// TwinCAT 3 PLC project Felber
// ProgramVersion: 3.1.4024.0
// libraries:
//   EfficientIO Communicator, * (EfficientIO)
//   EfficientIO Energy Basic, * (EfficientIO)
//   Lynus Persistent Data V1, * (Lynus AG)
//   Lynus Standards, * (EfficientIO)
//   Tc2_BABasic, * (Beckhoff Automation GmbH)
//   Tc2_EtherCAT, * (Beckhoff Automation GmbH)
//   Tc2_Standard, * (Beckhoff Automation GmbH)
//   Tc2_System, * (Beckhoff Automation GmbH)
//   Tc2_Utilities, * (Beckhoff Automation GmbH)
//   Tc3_IPCDiag, * (Beckhoff Automation GmbH)
//   Tc3_Module, * (Beckhoff Automation GmbH)
// project tree:
//   DUTs/ struct_ADS_Felber.TcDUT
//   ENUMs/ E_State.TcDUT
//   / FastTask.TcTTO (not stored), MiddleTask.TcTTO, SlowTask.TcTTO (not stored)
//   FBs/EL3443_DPM/DUTs/ E_EL3443_DPM_Phase.TcDUT (not stored), E_EL3443_DPM_Total.TcDUT (not stored), MDP5001_341_7CD731EE.TcDUT, MDP5001_341_I_7CD731EE.TcDUT (not stored), MDP5001_341_O_7CD731EE.TcDUT (not stored), ST_EL3443_DPM_MUX_REAL.TcDUT, ST_EL3443_DPM_MUX_ULINT.TcDUT, ST_EL3443_DPM_StatusLx.TcDUT, ST_EL3443_DPM_StatusTotal.TcDUT, ST_EL3443_DPM_VariantLx.TcDUT (not stored), ST_EL3443_DPM_VariantTotal.TcDUT (not stored), ST_EL3443_DPM_VariantValues.TcDUT
//   FBs/EL3443_DPM/ FB_EL3443_DPM.TcPOU
//   FBs/EL3446 FW02 or higher/DUTs/ E_EL3446_Phase.TcDUT, MDP5001_342_066CA8C6.TcDUT (not stored), MDP5001_342_I_066CA8C6.TcDUT (not stored), MDP5001_342_O_066CA8C6.TcDUT (not stored), ST_EL3446_MUX_REAL.TcDUT (not stored), ST_EL3446_MUX_ULINT.TcDUT, ST_EL3446_StatusIx.TcDUT, ST_EL3446_VariantIx.TcDUT, ST_EL3446_VariantValues.TcDUT
//   FBs/EL3446 FW02 or higher/ FB_EL3446.TcPOU (not stored)
//   FBs/ FB_CoE_EL3446.TcPOU, FB_CoE_EL3443.TcPOU, FB_EM_Beckhoff_EL3443.TcPOU, FB_EM_Beckhoff_EL3446.TcPOU, FB_TimeSwitch_V2.TcPOU (not stored), prg_ReadDeviceName.TcPOU (not stored)
//   POUs/ prgComEffIO.TcPOU, prgEM.TcPOU (not stored), prgEMS.TcPOU, prgHW_v1.TcPOU (not stored), prgPersistent.TcPOU, prgRWEffIO.TcPOU (not stored), prgSystemTime.TcPOU (not stored), prgVarEffIO.TcPOU (not stored)

CONFIGURATION Felber
    RESOURCE PLC ON TwinCAT3
        TASK MiddleTask(INTERVAL := T#10ms, PRIORITY := 22);
        PROGRAM prgPersistent WITH MiddleTask : prgPersistent;
        PROGRAM prgSystemTime WITH MiddleTask : prgSystemTime;
        PROGRAM prgEM WITH MiddleTask : prgEM;
        PROGRAM prgEMS WITH MiddleTask : prgEMS;
    END_RESOURCE
END_CONFIGURATION

// ---- DUTs/struct_ADS_Felber.TcDUT
TYPE struct_ADS_Felber :
STRUCT
	int_liveCount		: INT;	
	
	// prgEM
	lr_RealPower_Grid			: LREAL;				
	lr_ApparentPower_Grid		: LREAL;				
	lr_ReactivePower_Grid		: LREAL;				
	lr_Frequency_Grid			: LREAL;				                                   
	lr_Voltage_L1N				: LREAL;				
	lr_Voltage_L2N				: LREAL;				
	lr_Voltage_L3N				: LREAL;				
	lr_Voltage_L1L2				: LREAL;				
	lr_Voltage_L2L3				: LREAL;				
	lr_Voltage_L3L1				: LREAL;				
 	lr_Current_L1				: LREAL;				
	lr_Current_L2				: LREAL;				
	lr_Current_L3				: LREAL;				
	lrPower_EM1					: LREAL;					
	lrPower_EM2					: LREAL;					
	lrPower_EM3					: LREAL;					
	lrPower_EM4					: LREAL;					
	lrPower_EM5					: LREAL;					
	lrPower_EM6					: LREAL;					
	lrPower_House				: LREAL;					
	lr_EnergyCounter_Grid		: LREAL;					
	lr_EnergyCounter_EM1		: LREAL;					
	lr_EnergyCounter_EM2		: LREAL;					
	lr_EnergyCounter_EM3		: LREAL;					
	lr_EnergyCounter_EM4		: LREAL;					
	lr_EnergyCounter_EM5		: LREAL;					
	lr_EnergyCounter_EM6		: LREAL;					
	lr_EnergyCounter_House		: LREAL;		

	// prgEMS
	b_Manual_On_CH1				: BOOL;						
	b_Manual_Off_CH1			: BOOL;						
	b_Manual_On_CH2				: BOOL;						
	b_Manual_Off_CH2			: BOOL;						
	b_Manual_On_CH3				: BOOL;						
	b_Manual_Off_CH3			: BOOL;						
	b_Manual_On_CH4				: BOOL;						
	b_Manual_Off_CH4			: BOOL;						
	b_Manual_On_CH5				: BOOL;						
	b_Manual_Off_CH5			: BOOL;						
	b_Manual_On_Coffee_CH6		: BOOL;				
	b_Manual_Off_Coffee_CH6		: BOOL;				
	b_Manual_On_Vent_CH7		: BOOL;				
	b_Manual_Off_Vent_CH7		: BOOL;			
	b_LoadOn_CH1				: BOOL;		
	b_LoadOn_CH2				: BOOL;			
	b_LoadOn_CH3				: BOOL;			
	b_LoadOn_CH4				: BOOL;			
	b_LoadOn_CH5				: BOOL;			
	b_LoadOn_CH6				: BOOL;			
	b_LoadOn_CH7				: BOOL;		
	byte_MoFr_Open_Hour			: BYTE;					
	byte_MoFr_Open_Minute		: BYTE;					
	byte_MoFr_Close_Hour		: BYTE;					
	byte_MoFr_Close_Minute		: BYTE;					
	byte_Sa_Open_Hour			: BYTE;					
	byte_Sa_Open_Minute			: BYTE;					
	byte_Sa_Close_Hour			: BYTE;					
	byte_Sa_Close_Minute		: BYTE;					
	byte_So_Open_Hour			: BYTE;					
	byte_So_Open_Minute			: BYTE;					
	byte_So_Close_Hour			: BYTE;					
	byte_So_Close_Minute		: BYTE;					
// offset CH1 in hours			                    
	b_Enable_Control_CH1		: BOOL;				
	real_Offset_Start_CH1		: REAL;				
	real_Offset_Stop_CH1		: REAL;				
// offset CH2 in hours			                    
	b_Enable_Control_CH2		: BOOL;				
	real_Offset_Start_CH2		: REAL;				
	real_Offset_Stop_CH2		: REAL;				
// offset CH3 in hours			                    
	b_Enable_Control_CH3		: BOOL;				
	real_Offset_Start_CH3		: REAL;				
	real_Offset_Stop_CH3		: REAL;				
// offset CH4 in hours			                    
	b_Enable_Control_CH4		: BOOL;				
	real_Offset_Start_CH4		: REAL;				
	real_Offset_Stop_CH4		: REAL;				
// offset CH5 in hours			                    
	b_Enable_Control_CH5		: BOOL;				
	real_Offset_Start_CH5		: REAL;				
	real_Offset_Stop_CH5		: REAL;				
// offset CH6 in hours			                    
	b_Enable_Control_Coffee_CH6	: BOOL;				
	real_Offset_Start_Coffee_CH6: REAL;				
	real_Offset_Stop_Coffee_CH6	: REAL;				
// offset CH7 in hours			                    
	b_Enable_Control_Vent_CH7	: BOOL;				
	real_Offset_Start_CH7		: REAL;				
	real_Offset_Stop_CH7		: REAL;				


                                  
			(*: REAL;			                        
			: REAL;                                     
			: REAL;			
			: REAL;			
			: REAL;
			: REAL;			
			: REAL;
			: REAL;			
*)

END_STRUCT
END_TYPE

// ---- ENUMs/E_State.TcDUT
{attribute 'qualified_only'}
TYPE E_State :
(
	Init := 0,
	ReadOnce,
	Error,
	Idle,
	Wait

	
);
END_TYPE

// ---- FBs/EL3443_DPM/DUTs/MDP5001_341_7CD731EE.TcDUT
TYPE MDP5001_341_7CD731EE :
STRUCT
	MDP5001_341_Input	: MDP5001_341_I_7CD731EE;
	MDP5001_341_Output	: MDP5001_341_O_7CD731EE;
END_STRUCT
END_TYPE

// ---- FBs/EL3443_DPM/DUTs/ST_EL3443_DPM_MUX_REAL.TcDUT
TYPE ST_EL3443_DPM_MUX_REAL :
STRUCT
    nSelector : UINT := E_EL3443_DPM_Phase.Error_INDEX_Not_Valid;
    fValueRef : REFERENCE TO REAL;
END_STRUCT
END_TYPE

// ---- FBs/EL3443_DPM/DUTs/ST_EL3443_DPM_MUX_ULINT.TcDUT
TYPE ST_EL3443_DPM_MUX_ULINT :
STRUCT
    nSelector : UINT := E_EL3443_DPM_Phase.Error_INDEX_Not_Valid;
    nValueRef : POINTER TO ULINT;
END_STRUCT
END_TYPE

// ---- FBs/EL3443_DPM/DUTs/ST_EL3443_DPM_StatusLx.TcDUT
TYPE ST_EL3443_DPM_StatusLx :
STRUCT
    bStatus_Voltage_Sign_Bit : BOOL;             //Voltage Sign Bit - Indicates the sign of the current sine wave voltage: 1 = U > 0V, 0 = U < 0V
    bStatus_Overvoltage : BOOL;                  //Overvoltage - Maximum measurable voltage is exceeded.
    bStatus_Overcurrent : BOOL;                  //Overcurrent - Maximum measurable current is exceeded.
    bStatus_Inaccurate_Voltage : BOOL;           //Inaccurate Voltage - The measured voltage value is smaller than the value entered in CoE object "F800:15 Inaccurate Threshold Voltage".
    bStatus_Inaccurate_Current : BOOL;           //Inaccurate Current - The measured current value is smaller than the value entered in CoE object "F800:16 Inaccurate Threshold Current".
    bStatus_Voltage_Guard_Warning : BOOL;        //Voltage Guard Warning - A warning limit of the voltage monitor has been breached.
    bStatus_Voltage_Guard_Error : BOOL;          //Voltage Guard Error - An error limit of the voltage monitor has been breached.
    bStatus_Current_Guard_Warning : BOOL;        //Voltage Current Warning - A warning limit of the Current monitor has been breached.
    bStatus_Current_Guard_Error : BOOL;          //Voltage Current Error - An error limit of the Current monitor has been breached.
    bStatus_TxPDO_Toggle : BOOL;                 //TxPDO Toggle - The TxPDO toggle is toggled by the slave when the data of the associated TxPDO is updated.
END_STRUCT
END_TYPE

// ---- FBs/EL3443_DPM/DUTs/ST_EL3443_DPM_StatusTotal.TcDUT
TYPE ST_EL3443_DPM_StatusTotal :
STRUCT
    bStatus_System_State : BOOL;                         //System State - Overall system state (as a logical disjunction of voltage guard errors, phase sequence, overvoltage, overcurrent and frequency guard errors)
    bStatus_Grid_Direction : BOOL;                       //Grid Direction - Phase sequence L1 - L2 - L3 correctly detected (with clockwise 3-phase mains)
    bStatus_Frequency_Guard_Warning : BOOL;              //Frequency Guard Warning - A warning limit of the frequency monitor has been breached.
    bStatus_Frequency_Guard_Error : BOOL;                //Frequency Guard Error - An error limit of the frequency monitor has been breached.
    bStatus_Neutral_Current_Guard_Warning : BOOL;        //Neutral Current Guard Warning - A warning limit of the neutral conductor current monitor has been breached.
    bStatus_Neutral_Current_Guard_Error : BOOL;          //Neutral Current Guard Error - An error limit of the neutral conductor current monitor has been breached.
    bStatus_Active_Power_Guard_Warning : BOOL;           //Active Power Guard Warning - A warning limit of the active power monitor has been breached.
    bStatus_Active_Power_Guard_Error : BOOL;             //Active Power Guard Error - An error limit of the active power monitor has been breached.
    bStatus_Apparent_Power_Guard_Warning : BOOL;         //Apparent Power Guard Warning - A warning limit of the apparent power monitor has been breached.
    bStatus_Apparent_Power_Guard_Error : BOOL;           //Apparent Power Guard Error - An error limit of the apparent power monitor has been breached.
    bStatus_Power_Quality_Guard_Warning : BOOL;          //Power Quality Guard Warning - A warning limit of the PQF monitor has been breached.
    bStatus_Power_Quality_Guard_Error : BOOL;            //Power Quality Guard Error - An error limit of the PQF monitor has been breached.
    bStatus_TxPDO_State : BOOL;                          //TxPDO State - TRUE for general error
    bStatus_TxPDO_Toggle : BOOL;                         //TxPDO Toggle - The TxPDO toggle is toggled by the slave when the data of the associated TxPDO is updated.
    fStatus_Power_Quality_Factor : REAL;                 //Power Quality Factor - Analog value of the voltage quality between 1.0 and 0 (see basic function principles - Power Quality Factor)
END_STRUCT                                              
END_TYPE

// ---- FBs/EL3443_DPM/DUTs/ST_EL3443_DPM_VariantValues.TcDUT
{attribute 'no-analysis'}
TYPE ST_EL3443_DPM_VariantValues :
STRUCT
	astLx 			: ARRAY[1..3] OF ST_EL3443_DPM_VariantLx;
	stTotal 		: ST_EL3443_DPM_VariantTotal;
END_STRUCT
END_TYPE

// ---- FBs/EL3446 FW02 or higher/DUTs/E_EL3446_Phase.TcDUT
(*This enum is equivalent to the selectors from the documentation " Confirmation of variable output values 1 - 4"*)
{attribute 'qualified_only'}
TYPE E_EL3446_Phase :
(
    nPhaseI1_OFFSET := 256,     //Offset Channel 1(Current I1). The offset is added to the base selector     
    nPhaseI2_OFFSET := 512,     //Offset Channel 2(Current I2). The offset is added to the base selector
    nPhaseI3_OFFSET := 768,     //Offset Channel 3(Current I3). The offset is added to the base selector
    nPhaseI4_OFFSET := 1024,    //Offset Channel 4(Current I1). The offset is added to the base selector     
    nPhaseI5_OFFSET := 1280,    //Offset Channel 5(Current I2). The offset is added to the base selector
    nPhaseI6_OFFSET := 1536,    //Offset Channel 6(Current I3). The offset is added to the base selector
    
    
    U_RMS:= 1,                  // [V] (Real Selector: 1 (Examp.: 257 = 1 + 256 for ch. 1)) RMS value of the voltage
    I_RMS:= 8,                  // [A] (Real Selector: 8) RMS value of the current 
	Frequency:= 17,             // [Hz] (Real Selector: 17) Frequency of this phase
    Phi:= 21,                   // [°] (Real Selector: 21) Phase angle of the fundamental wave
    Cos_phi:= 22,               // [-] (Real Selector: 22) Cosine of the fundamental wave phase angle
    Power_Factor:= 23,          // [-] (Real Selector: 23) Power factor
    P:= 26,                     // [W] (Real Selector: 26) Active power
	(*available with FW02 and higher*) Pavg := 27,                 // [W] (Real Selector: 27) Average active power during the last interval
	(*available with FW02 and higher*) Pmin := 28,                 // [W] (Real Selector: 28) Minimum active power in the last interval
	(*available with FW02 and higher*) Pmax := 29,                 // [W] (Real Selector: 29) Maximum active power in the last interval
	Pfund:= 30,					// [W] (Real Selector: 30) Fundamental wave active power in the last interval
    S_:= 32,                    // [VA] (Real Selector: 32) Apparent power
	(*available with FW02 and higher*) Savg := 33,                 // [W] (Real Selector: 33) Average apparent power during the last interval
	(*available with FW02 and higher*) Smin := 34,                 // [W] (Real Selector: 34) Minimum apparent power in the last interval
	(*available with FW02 and higher*) Smax := 35,                 // [W] (Real Selector: 35) Maximum apparent power in the last interval
	Sfund:= 36,					// [VA] (Real Selector: 36) Fundamental wave apparent power in the last interval
    Q:= 38,                     // [Var] (Real Selector: 38) Reactive power
	(*available with FW02 and higher*) Qavg := 39,                 // [W] (Real Selector: 39) Average reactive power during the last interval
	(*available with FW02 and higher*) Qmin := 40,                 // [W] (Real Selector: 40) Minimum reactive power in the last interval
	(*available with FW02 and higher*) Qmax := 41,                 // [W] (Real Selector: 41) Maximum reactive power in the last interval
	Qfund:= 42,					// [Var] (Real Selector: 36) Fundamental wave reactive power in the last interval
    EP:= 45,                    // [mhW] (UINT Selector: 45) Recorded active energy
    EP_pos:= 46,                // [mhW] (UINT Selector: 46) Received active energy
    EP_neg:= 47,                // [mhW] (UINT Selector: 47) Supplied active energy
	EP_interval:= 48, 			// [mhW] (UINT Selector: 48) Recorded active energy in the last interval
	EP_pos_interval:= 49, 		// [mhW] (UINT Selector: 49) Received active energy in the last interval
	EP_neg_interval:= 50, 		// [mhW] (UINT Selector: 50) Supplied active energy in the last interval
    ES:= 51,                    // [mhW] (UINT Selector: 51) Apparent energy
    ES_pos:= 52,                // [mhW] (UINT Selector: 52) Apparent energy
    ES_neg:= 53,                // [mhW] (UINT Selector: 53) Apparent energy
	ES_interval:= 54, 			// [mhW] (UINT Selector: 54) Apparent energy in the last interval
	ES_pos_interval:= 55, 		// [mhW] (UINT Selector: 55) Apparent energy in the last interval
	ES_neg_interval:= 56, 		// [mhW] (UINT Selector: 56) Apparent energy in the last interval
    EQ_:= 57,                   // [mhW] (UINT Selector: 57) Reactive energy
    EQ_pos:= 58,                // [mhW] (UINT Selector: 58) Reactive energy
    EQ_neg:= 59,                // [mhW] (UINT Selector: 59) Reactive energy
	EQ_interval:= 60, 			// [mhW] (UINT Selector: 60) Reactive energy in the last interval
	EQ_pos_interval:= 61, 		// [mhW] (UINT Selector: 62) Reactive energy in the last interval
	EQ_neg_interval:= 62, 		// [mhW] (UINT Selector: 63) Reactive energy in the last interval
    THD_U:= 95,                 // [-] (Real Selector: 95) "Total Harmonic Distortion" is the distortion factor of the voltage. It indicates the ratio of the harmonic components of an oscillation relative to its fundamental.
    RMS_fund_U:= 98,            // [V] (Real Selector: 98) Amplitude of the fundamental wave
	THD_I:= 165,                // [-] (Real Selector: 165) "Total Harmonic Distortion" is the distortion factor of the current. It indicates the ratio of the harmonic components of an oscillation relative to its fundamental.
    RMS_fund_I:= 168,           // [A] (Real Selector: 168) Amplitude of the fundamental wave
    (*available with FW02 and higher*) F_Ref_I:= 169,              // [Hz] (Real Selector: 169) Reference frequency of the current harmonic: Specifies the underlying fundamental frequency, e.g.: 50 or 60 Hz.
    Harmonics_I := 170,         // [% of the fundamental wave] (Real Selector: 170-211) 0 => DC component, 1 => fundamental wave, 2=> 2nd harmonic, 3=> 3rd harmonic
    Error_INDEX_Not_Valid:= 255 // [-] (Real Selector: 255) Error message: The selected index is not available.
)UINT;
END_TYPE

// ---- FBs/EL3446 FW02 or higher/DUTs/ST_EL3446_MUX_ULINT.TcDUT
TYPE ST_EL3446_MUX_ULINT :
STRUCT
    nSelector : UINT := E_EL3446_Phase.Error_INDEX_Not_Valid;
    nValueRef : POINTER TO ULINT;
END_STRUCT
END_TYPE

// ---- FBs/EL3446 FW02 or higher/DUTs/ST_EL3446_StatusIx.TcDUT
TYPE ST_EL3446_StatusIx :
STRUCT
	bOvercurrent : BOOL;                    //Overcurrent - Maximum measurable current is exceeded.
	bInaccurate_Current : BOOL;             //Inaccurate Current - The measured current value is outside the limits for the current entered in CoE object 0x80n2
	bCurrent_Guard_Warning : BOOL;          //Current Guard Warning - The measured current value is outside the warning limits entered in the CoE objects 0x80n2:06 and 0x80n2:07
	bCurrent_Guard_Error : BOOL;            //Current Guard Error - The measured current value is outside the error limits entered in the CoE objects 0x80n2:05 and 0x80n2:08
	bApparent_Power_Guard_Warning : BOOL;   //Apparent Power Guard Warning - The value for the apparent power is outside the warning limits entered in the CoE objects 0x80n2:0A and 0x80n2:0B
	bApparent_Power_Guard_Error : BOOL;     //Apparent Power Guard Error - The value for the apparent power is outside the error limits for the current entered in the CoE objects 0x80n2:09 and 0x80n2:0C
	bActive_Power_Guard_Warning : BOOL;     //Active Power Guard Warning - The value for active power is outside the warning limits entered in the CoE objects 0x80n2:0E and 0x80n2:0F
	bActive_Power_Guard_Error : BOOL;       //Active Power Guard Error - The value for active power is outside the error limits for the current entered in CoE objects 0x80n2:0D and 0x80n2:10
	bReactive_Power_Guard_Warning : BOOL;   //Reactive Power Guard Warning - The value for the reactive power is outside the warning limits entered in the CoE objects 0x80n2:12 and 0x80n2:13
	bReactive_Power_Guard_Error : BOOL;     //Reactive Power Guard Error - The value for the reactive power is outside the error limits for the current entered in the CoE objects 0x80n2:11 and 0x80n2:14
	bDPM_Inaccurate : BOOL;                 //DPM Inaccurate
	bDPM_Timeout : BOOL;                    //DPM Toggl e- The DPM toggle is toggled by the slave when the DPM data has been updated.
	bTxPDO_Toggle : BOOL;                   //TxPDO Toggle - The TxPDO toggle is toggled by the slave when the data of the associated TxPDO has been updated.
	fCurrent : REAL;                        //Current - Actual measured current value
	fActive_Power : REAL;                   //Active Power - Actually measured active power
	fApparent_Power : REAL;                 //Apparent Power - Actual measured apparent power
	fReactive_Power_Fundamental : REAL;     //Reactive Power Fundamental - Balanced reactive power fundamental oscillation
	nActive_Energy : DINT;                  //Active Energy - Actually measured active energy
END_STRUCT
END_TYPE

// ---- FBs/EL3446 FW02 or higher/DUTs/ST_EL3446_VariantIx.TcDUT
TYPE ST_EL3446_VariantIx :
STRUCT
    fU_RMS : REAL;// [V] (Real Selector: 1 (Examp.: 257 = 1 + 256 for ch. 1)) RMS value of the voltage
    fI_RMS : REAL;// [A] (Real Selector: 8) RMS value of the current
    fFrequency : REAL;// [Hz] (Real Selector: 17) Frequency of this phase
    fPhi : REAL;// [°] (Real Selector: 21) Phase angle of the fundamental wave
    fCOS_phi : REAL;// [-] (Real Selector: 22) Cosine of the fundamental wave phase angle
    fPower_Factor : REAL;// [-] (Real Selector: 23) Power factor
    fP : REAL;// [W] (Real Selector: 26) Active power
	(*available with FW02 and higher*) fPavg : REAL;						// [W] (Real Selector: 27) Average active power during the last interval
    (*available with FW02 and higher*) fPmin : REAL;						// [W] (Real Selector: 28) Minimum active power in the last interval
    (*available with FW02 and higher*) fPmax : REAL;						// [W] (Real Selector: 29) Maximum active power in the last interval
	fPfund : REAL;// [W] (Real Selector: 30) Fundamental wave active power in the last interval
	fS : REAL;// [VA] (Real Selector: 32) Apparent power
	(*available with FW02 and higher*) fSavg : REAL;						// [VA] (Real Selector: 33) Average apparent power during the last interval
    (*available with FW02 and higher*) fSmin : REAL;						// [VA] (Real Selector: 34) Minimum apparent power in last interval
   	(*available with FW02 and higher*) fSmax : REAL;						// [VA] (Real Selector: 35) Minimum apparent power in last interval
    fSfund : REAL;// [VA] (Real Selector: 36) Fundamental wave apparent power in the last interval
    fQ : REAL;// [Var] (Real Selector: 38) Reactive power
	(*available with FW02 and higher*) fQavg : REAL;						// [Var] (Real Selector: 39) Average reactive power average during the last interval
    (*available with FW02 and higher*) fQmin : REAL;						// [Var] (Real Selector: 40) Minimum reactive power in the last interval
    (*available with FW02 and higher*) fQmax : REAL;						// [Var] (Real Selector: 41) Maximum reactive power in the last interval
    fQfund : REAL;// [Var] (Real Selector: 42) Fundamental wave reactive power in the last interval
    nEP : LINT;// [mhW] (LINT Selector: 45) Recorded active energy
    nEP_pos : ULINT;// [mhW] (UINT Selector: 46) Received active energy
    nEP_neg : ULINT;// [mhW] (UINT Selector: 47) Supplied active energy
	nEP_interval : LINT;// [mhW] (LINT Selector: 48) Recorded active energy in the last interval
	nEP_pos_interval : ULINT;// [mhW] (UINT Selector: 49) Received active energy in the last interval
	nEP_neg_interval : ULINT;// [mhW] (UINT Selector: 50) Supplied active energy in the last interval
    nES : LINT;// [mhW] (LINT Selector: 51) Apparent energy
    nES_pos : ULINT;// [mhW] (UINT Selector: 52) Apparent energy
    nES_neg : ULINT;// [mhW] (UINT Selector: 53) Apparent energy
	nES_interval : LINT;// [mhW] (LINT Selector: 54) Apparent energy in the last interval
	nES_pos_interval : ULINT;// [mhW] (UINT Selector: 55) Apparent energy in the last interval
	nES_neg_interval : ULINT;// [mhW] (UINT Selector: 56) Apparent energy in the last interval
    nEQ : LINT;// [mhW] (LINT Selector: 57) Reactive energy
    nEQ_pos : ULINT;// [mhW] (UINT Selector: 58) Reactive energy
    nEQ_neg : ULINT;// [mhW] (UINT Selector: 59) Reactive energy
	nEQ_interval : LINT;// [mhW] (LINT Selector: 60) Reactive energy in the last interval
	nEQ_pos_interval : ULINT;// [mhW] (UINT Selector: 62) Reactive energy in the last interval
	nEQ_neg_interval : ULINT;// [mhW] (UINT Selector: 63) Reactive energy in the last interval
    fTHD_U : REAL;// [-] (Real Selector: 95) "Total Harmonic Distortion" is the distortion factor of the voltage. It indicates the ratio of the harmonic components of an oscillation relative to its fundamental.
    fRMS_fund_U : REAL;// [V] (Real Selector: 98) Amplitude of the fundamental wave
    fTHD_I : REAL;// [-] (Real Selector: 165) "Total Harmonic Distortion" is the distortion factor of the current. It indicates the ratio of the harmonic components of an oscillation relative to its fundamental.
    fRMS_fund_I : REAL;// [A] (Real Selector: 168) Amplitude of the fundamental wave
    (*available with FW02 and higher*) fF_Ref_I : REAL;// [Hz] (Real Selector: 169) Reference frequency of the current harmonic: Specifies the underlying fundamental frequency, e.g.: 50 or 60 Hz.
    fHarmonics_I : ARRAY [0..41] OF REAL;// [% of the fundamental wave] (Real Selector: 170-211) 0 => DC component, 1 => fundamental wave, 2=> 2nd harmonic, 3=> 3rd harmonic
END_STRUCT
END_TYPE

// ---- FBs/EL3446 FW02 or higher/DUTs/ST_EL3446_VariantValues.TcDUT
{attribute 'no-analysis'}
TYPE ST_EL3446_VariantValues :
STRUCT
	astIx 			: ARRAY[1..6] OF ST_EL3446_VariantIx;
END_STRUCT
END_TYPE

// ---- POUs/prgPersistent.TcPOU
PROGRAM prgPersistent
VAR
	fbUSV		: FB_WritePersistentData_CX81xx;

	fb_Reboot		: NT_reboot;
	m_Reboot		: BOOL:=FALSE;
END_VAR

fbUSV(
	eSaveModeData:= eUSVSaveMode.eSaveWhenPowerfail, 
	bLoadPersistentDataOk=> , 
	bPowerFailDetect=> , 
	bError=> , 
	bySaveProcess=> , 
	dwStorageLast24h=> , 
	udiErrorCode=> );
	
	
		
fb_Reboot(	netid := '',
			delay := 2,
			start := m_Reboot);

END_PROGRAM

// ---- POUs/prgEMS.TcPOU
PROGRAM prgEMS
VAR
	FB_TimeSwitch_CH1: FB_TimeSwitch_v2;
	FB_TimeSwitch_CH2: FB_TimeSwitch_v2;
	FB_TimeSwitch_CH3: FB_TimeSwitch_v2;
	FB_TimeSwitch_CH4: FB_TimeSwitch_v2;
	FB_TimeSwitch_CH5: FB_TimeSwitch_v2;	// outside light
	FB_TimeSwitch_CH6: FB_TimeSwitch_v2;	// Coffee maschine
	FB_TimeSwitch_CH7: FB_TimeSwitch_v2;	// Ventilation
	FB_TimeSwitch_CH8: FB_TimeSwitch_v2;	// Coffee maschine2
	TEST				:MDP5001_341_224AC5A3;
	b_Manual_On_CH1		: BOOL;						//{#lynus.ag#()}
	b_Manual_Off_CH1	: BOOL;						//{#lynus.ag#()}
	b_Manual_On_CH2		: BOOL;						//{#lynus.ag#()}
	b_Manual_Off_CH2	: BOOL;						//{#lynus.ag#()}
	b_Manual_On_CH3		: BOOL;						//{#lynus.ag#()}
	b_Manual_Off_CH3	: BOOL;						//{#lynus.ag#()}
	b_Manual_On_CH4		: BOOL;						//{#lynus.ag#()}
	b_Manual_Off_CH4	: BOOL;						//{#lynus.ag#()}
	b_Manual_On_CH5		: BOOL;						//{#lynus.ag#()}
	b_Manual_Off_CH5	: BOOL;						//{#lynus.ag#()}
	b_Manual_On_Coffee_CH6		: BOOL;						//{#lynus.ag#()}
	b_Manual_Off_Coffee_CH6		: BOOL;						//{#lynus.ag#()}
	b_Manual_On_Vent_CH7		: BOOL;						//{#lynus.ag#()}
	b_Manual_Off_Vent_CH7		: BOOL;						//{#lynus.ag#()}
	b_Manual_On_Coffee2_CH8		: BOOL;						//{#lynus.ag#()}
	b_Manual_Off_Coffee2_CH8	: BOOL;						//{#lynus.ag#()}

	fbCalcSunriseSunset   		: FB_CalcSunriseSunset;
	todSunrise            		: TOD;
	todSunset             		: TOD;
	fb_GetTimeZoneInfo	:FB_GetTimeZoneInformation;
	b_firstCycle: BOOL;
	RS_Outsidelight: RS;
	r_trig_on: R_trig;
	r_trig_off: R_trig;
	b_Out_CH1: BOOL;
	b_Out_CH2: BOOL;
	b_Out_CH3: BOOL;
	b_Out_CH4: BOOL;
	b_Out_CH5: BOOL;
	b_Out_CH6: BOOL;
	b_Out_CH7: BOOL;		
	b_Out_CH8: BOOL;		
	b_LoadOn_CH1	: BOOL;						//{#lynus.ag#()}
	b_LoadOn_CH2	: BOOL;						//{#lynus.ag#()}
	b_LoadOn_CH3	: BOOL;						//{#lynus.ag#()}
	b_LoadOn_CH4	: BOOL;						//{#lynus.ag#()}
	b_LoadOn_CH5	: BOOL;						//{#lynus.ag#()}
	b_LoadOn_CH6	: BOOL;						//{#lynus.ag#()}
	b_LoadOn_CH7	: BOOL;						//{#lynus.ag#()}
	b_LoadOn_CH8	: BOOL;						//{#lynus.ag#()}
END_VAR
VAR_INPUT
	fDegreeOfLongitude 	:LREAL;
	fDegreeOfLatitude	:LREAL;
	b_Input_KeySwitch		: BOOL;						//{#lynus.ag#()}
	b_Input_Spare			: BOOL;						//{#lynus.ag#()}
	m_UnderGroundMode		: BOOL;						//{#lynus.ag#()}
	int_test:INT;
END_VAR
VAR PERSISTENT
// opening hours
	byte_MoFr_Open_Hour		:BYTE;					//{#lynus.ag#()}
	byte_MoFr_Open_Minute	:BYTE;					//{#lynus.ag#()}
	byte_MoFr_Close_Hour	:BYTE;					//{#lynus.ag#()}
	byte_MoFr_Close_Minute	:BYTE;					//{#lynus.ag#()}
	byte_Sa_Open_Hour		:BYTE;					//{#lynus.ag#()}
	byte_Sa_Open_Minute		:BYTE;					//{#lynus.ag#()}
	byte_Sa_Close_Hour		:BYTE;					//{#lynus.ag#()}
	byte_Sa_Close_Minute	:BYTE;					//{#lynus.ag#()}
	byte_So_Open_Hour		:BYTE;					//{#lynus.ag#()}
	byte_So_Open_Minute		:BYTE;					//{#lynus.ag#()}
	byte_So_Close_Hour		:BYTE;					//{#lynus.ag#()}
	byte_So_Close_Minute	:BYTE;					//{#lynus.ag#()}
// offset CH1 in hours			
	b_Enable_Control_CH1		:BOOL;				//{#lynus.ag#()}
	real_Offset_Start_CH1		:REAL;				//{#lynus.ag#()}
	real_Offset_Stop_CH1		:REAL;				//{#lynus.ag#()}
// offset CH2 in hours			
	b_Enable_Control_CH2		:BOOL;				//{#lynus.ag#()}
	real_Offset_Start_CH2		:REAL;				//{#lynus.ag#()}
	real_Offset_Stop_CH2		:REAL;				//{#lynus.ag#()}
// offset CH3 in hours			
	b_Enable_Control_CH3		:BOOL;				//{#lynus.ag#()}
	real_Offset_Start_CH3		:REAL;				//{#lynus.ag#()}
	real_Offset_Stop_CH3		:REAL;				//{#lynus.ag#()}
// offset CH4 in hours			
	b_Enable_Control_CH4		:BOOL;				//{#lynus.ag#()}
	real_Offset_Start_CH4		:REAL;				//{#lynus.ag#()}
	real_Offset_Stop_CH4		:REAL;				//{#lynus.ag#()}
// offset CH5 in hours			
	b_Enable_Control_CH5		:BOOL;				//{#lynus.ag#()}
	real_Offset_Start_CH5		:REAL;				//{#lynus.ag#()}
	real_Offset_Stop_CH5		:REAL;				//{#lynus.ag#()}
// offset CH6 in hours			
	b_Enable_Control_Coffee_CH6	:BOOL;				//{#lynus.ag#()}
	real_Offset_Start_Coffee_CH6:REAL;				//{#lynus.ag#()}
	real_Offset_Stop_Coffee_CH6	:REAL;				//{#lynus.ag#()}
// offset CH7 in hours			
	b_Enable_Control_Vent_CH7	:BOOL;				//{#lynus.ag#()}
	real_Offset_Start_CH7		:REAL;				//{#lynus.ag#()}
	real_Offset_Stop_CH7		:REAL;				//{#lynus.ag#()}
// offset CH8 in hours			
	b_Enable_Control_Coffee2_CH8	:BOOL;				//{#lynus.ag#()}
	real_Offset_Start_Coffee2_CH8	:REAL;				//{#lynus.ag#()}
	real_Offset_Stop_Coffee2_CH8	:REAL;				//{#lynus.ag#()}
END_VAR


FB_TimeSwitch_CH1(
	b_Enable:= b_Enable_Control_CH1, 
	b_StatusOn:= NOT b_Out_CH1, 
	structSystemTime:=prgSystemTime.structSystemTime , 
	byte_MoFr_Open_Hour:= byte_MoFr_Open_Hour , 
	byte_MoFr_Open_Minute:= byte_MoFr_Open_Minute, 
	byte_MoFr_Close_Hour:= byte_MoFr_Close_Hour , 
	byte_MoFr_Close_Minute:= byte_MoFr_Close_Minute, 
	byte_Sa_Open_Hour:= byte_Sa_Open_Hour, 
	byte_Sa_Open_Minute:= byte_Sa_Open_Minute , 
	byte_Sa_Close_Hour:= byte_Sa_Close_Hour , 
	byte_Sa_Close_Minute:= byte_Sa_Close_Minute, 
	byte_So_Open_Hour:= byte_So_Open_Hour, 
	byte_So_Open_Minute:= byte_So_Open_Minute, 
	byte_So_Close_Hour:= byte_So_Close_Hour, 
	byte_So_Close_Minute:= byte_So_Close_Minute, 
	real_Offset_Start:= real_Offset_Start_CH1 , 
	real_Offset_Stop:= real_Offset_Stop_CH1 , 
	b_On_Manual:= b_Manual_On_CH1, 
	b_Off_Manual:= b_Manual_Off_CH1, 
	b_Output_On=> b_LoadOn_CH1, 
	b_Error=> );
b_Out_CH1 := NOT FB_TimeSwitch_CH1.b_Output_On;

FB_TimeSwitch_CH2(
	b_Enable:= b_Enable_Control_CH2, 
	b_StatusOn:= NOT b_Out_CH2, 
	structSystemTime:=prgSystemTime.structSystemTime , 
	byte_MoFr_Open_Hour:= byte_MoFr_Open_Hour , 
	byte_MoFr_Open_Minute:= byte_MoFr_Open_Minute, 
	byte_MoFr_Close_Hour:= byte_MoFr_Close_Hour , 
	byte_MoFr_Close_Minute:= byte_MoFr_Close_Minute, 
	byte_Sa_Open_Hour:= byte_Sa_Open_Hour, 
	byte_Sa_Open_Minute:= byte_Sa_Open_Minute , 
	byte_Sa_Close_Hour:= byte_Sa_Close_Hour , 
	byte_Sa_Close_Minute:= byte_Sa_Close_Minute, 
	byte_So_Open_Hour:= byte_So_Open_Hour, 
	byte_So_Open_Minute:= byte_So_Open_Minute, 
	byte_So_Close_Hour:= byte_So_Close_Hour, 
	byte_So_Close_Minute:= byte_So_Close_Minute, 
	real_Offset_Start:= real_Offset_Start_CH2 , 
	real_Offset_Stop:= real_Offset_Stop_CH2 , 
	b_On_Manual:= b_Manual_On_CH2, 
	b_Off_Manual:= b_Manual_Off_CH2, 
	b_Output_On=> b_LoadOn_CH2, 
	b_Error=> );
b_Out_CH2 := NOT FB_TimeSwitch_CH2.b_Output_On;

FB_TimeSwitch_CH3(
	b_Enable:= b_Enable_Control_CH3, 
	b_StatusOn:= NOT b_Out_CH3, 
	structSystemTime:=prgSystemTime.structSystemTime , 
	byte_MoFr_Open_Hour:= byte_MoFr_Open_Hour , 
	byte_MoFr_Open_Minute:= byte_MoFr_Open_Minute, 
	byte_MoFr_Close_Hour:= byte_MoFr_Close_Hour , 
	byte_MoFr_Close_Minute:= byte_MoFr_Close_Minute, 
	byte_Sa_Open_Hour:= byte_Sa_Open_Hour, 
	byte_Sa_Open_Minute:= byte_Sa_Open_Minute , 
	byte_Sa_Close_Hour:= byte_Sa_Close_Hour , 
	byte_Sa_Close_Minute:= byte_Sa_Close_Minute, 
	byte_So_Open_Hour:= byte_So_Open_Hour, 
	byte_So_Open_Minute:= byte_So_Open_Minute, 
	byte_So_Close_Hour:= byte_So_Close_Hour, 
	byte_So_Close_Minute:= byte_So_Close_Minute, 
	real_Offset_Start:= real_Offset_Start_CH3 , 
	real_Offset_Stop:= real_Offset_Stop_CH3 , 
	b_On_Manual:= b_Manual_On_CH3, 
	b_Off_Manual:= b_Manual_Off_CH3, 
	b_Output_On=> b_LoadOn_CH3, 
	b_Error=> );
b_Out_CH3 := NOT FB_TimeSwitch_CH3.b_Output_On;
	
FB_TimeSwitch_CH4(
	b_Enable:= b_Enable_Control_CH4, 
	b_StatusOn:= NOT b_Out_CH4, 
	structSystemTime:=prgSystemTime.structSystemTime , 
	byte_MoFr_Open_Hour:= byte_MoFr_Open_Hour , 
	byte_MoFr_Open_Minute:= byte_MoFr_Open_Minute, 
	byte_MoFr_Close_Hour:= byte_MoFr_Close_Hour , 
	byte_MoFr_Close_Minute:= byte_MoFr_Close_Minute, 
	byte_Sa_Open_Hour:= byte_Sa_Open_Hour, 
	byte_Sa_Open_Minute:= byte_Sa_Open_Minute , 
	byte_Sa_Close_Hour:= byte_Sa_Close_Hour , 
	byte_Sa_Close_Minute:= byte_Sa_Close_Minute, 
	byte_So_Open_Hour:= byte_So_Open_Hour, 
	byte_So_Open_Minute:= byte_So_Open_Minute, 
	byte_So_Close_Hour:= byte_So_Close_Hour, 
	byte_So_Close_Minute:= byte_So_Close_Minute, 
	real_Offset_Start:= real_Offset_Start_CH4 , 
	real_Offset_Stop:= real_Offset_Stop_CH4 , 
	b_On_Manual:= b_Manual_On_CH4, 
	b_Off_Manual:= b_Manual_Off_CH4, 
	b_Output_On=> b_LoadOn_CH4 ,
	b_Error=> );
b_Out_CH4 := NOT FB_TimeSwitch_CH4.b_Output_On;
	
FB_TimeSwitch_CH5(
	b_Enable:= b_Enable_Control_CH5, 
	b_StatusOn:= NOT b_Out_CH5, 
	structSystemTime:=prgSystemTime.structSystemTime , 
	byte_MoFr_Open_Hour:= byte_MoFr_Open_Hour , 
	byte_MoFr_Open_Minute:= byte_MoFr_Open_Minute, 
	byte_MoFr_Close_Hour:= byte_MoFr_Close_Hour , 
	byte_MoFr_Close_Minute:= byte_MoFr_Close_Minute, 
	byte_Sa_Open_Hour:= byte_Sa_Open_Hour, 
	byte_Sa_Open_Minute:= byte_Sa_Open_Minute , 
	byte_Sa_Close_Hour:= byte_Sa_Close_Hour , 
	byte_Sa_Close_Minute:= byte_Sa_Close_Minute, 
	byte_So_Open_Hour:= byte_So_Open_Hour, 
	byte_So_Open_Minute:= byte_So_Open_Minute, 
	byte_So_Close_Hour:= byte_So_Close_Hour, 
	byte_So_Close_Minute:= byte_So_Close_Minute, 
	real_Offset_Start:= real_Offset_Start_CH5 , 
	real_Offset_Stop:= real_Offset_Stop_CH5 , 
	b_On_Manual:= b_Manual_On_CH5, 
	b_Off_Manual:= b_Manual_Off_CH5, 
	b_Output_On=>  , 
	b_Error=> );
//b_Out_CH5 := NOT FB_TimeSwitch_CH5.b_Output_On; 		Outside light, done below
	
FB_TimeSwitch_CH6(
	b_Enable:= b_Enable_Control_Coffee_CH6, 
	b_StatusOn:= NOT b_Out_CH6, 
	structSystemTime:=prgSystemTime.structSystemTime , 
	byte_MoFr_Open_Hour:= byte_MoFr_Open_Hour , 
	byte_MoFr_Open_Minute:= byte_MoFr_Open_Minute, 
	byte_MoFr_Close_Hour:= byte_MoFr_Close_Hour , 
	byte_MoFr_Close_Minute:= byte_MoFr_Close_Minute, 
	byte_Sa_Open_Hour:= byte_Sa_Open_Hour, 
	byte_Sa_Open_Minute:= byte_Sa_Open_Minute , 
	byte_Sa_Close_Hour:= byte_Sa_Close_Hour , 
	byte_Sa_Close_Minute:= byte_Sa_Close_Minute, 
	byte_So_Open_Hour:= byte_So_Open_Hour, 
	byte_So_Open_Minute:= byte_So_Open_Minute, 
	byte_So_Close_Hour:= byte_So_Close_Hour, 
	byte_So_Close_Minute:= byte_So_Close_Minute, 
	real_Offset_Start:= real_Offset_Start_Coffee_CH6 , 
	real_Offset_Stop:= real_Offset_Stop_Coffee_CH6 , 
	b_On_Manual:= b_Manual_On_Coffee_CH6, 
	b_Off_Manual:= b_Manual_Off_Coffee_CH6, 
	b_Output_On=> b_LoadOn_CH6, 
	b_Error=> );
b_Out_CH6 := NOT FB_TimeSwitch_CH6.b_Output_On;
	
FB_TimeSwitch_CH7(
	b_Enable:= b_Enable_Control_Vent_CH7, 
	b_StatusOn:= NOT b_Out_CH7, 
	structSystemTime:=prgSystemTime.structSystemTime , 
	byte_MoFr_Open_Hour:= byte_MoFr_Open_Hour , 
	byte_MoFr_Open_Minute:= byte_MoFr_Open_Minute, 
	byte_MoFr_Close_Hour:= byte_MoFr_Close_Hour , 
	byte_MoFr_Close_Minute:= byte_MoFr_Close_Minute, 
	byte_Sa_Open_Hour:= byte_Sa_Open_Hour, 
	byte_Sa_Open_Minute:= byte_Sa_Open_Minute , 
	byte_Sa_Close_Hour:= byte_Sa_Close_Hour , 
	byte_Sa_Close_Minute:= byte_Sa_Close_Minute, 
	byte_So_Open_Hour:= byte_So_Open_Hour, 
	byte_So_Open_Minute:= byte_So_Open_Minute, 
	byte_So_Close_Hour:= byte_So_Close_Hour, 
	byte_So_Close_Minute:= byte_So_Close_Minute, 
	real_Offset_Start:= real_Offset_Start_CH7 , 
	real_Offset_Stop:= real_Offset_Stop_CH7 , 
	b_On_Manual:= b_Manual_On_Vent_CH7, 
	b_Off_Manual:= b_Manual_Off_Vent_CH7, 
	b_Output_On=> b_LoadOn_CH7, 
	b_Error=> );
b_Out_CH7 := NOT FB_TimeSwitch_CH7.b_Output_On;
	
	
// calculate sunset / sunrise
// find out the time details	
IF fDegreeOfLongitude= 0 OR fDegreeOfLatitude= 0 THEN 
	fDegreeOfLongitude := 16.3731;   (* Longitude of Vienna *)
	fDegreeOfLatitude := 48.2083;   (* Latitude of Vienna*)
END_IF
fb_GetTimeZoneInfo(
	sNetID:= '', 
	bExecute:= prgSystemTime.structSystemTime.wHour = 4 OR NOT b_firstCycle, 
	tTimeout:= T#5S, 
	bBusy=> , 
	bError=> , 
	nErrID=> , 
	tzID=> , 
	tzInfo=> );
b_firstCycle := TRUE;


fbCalcSunriseSunset(
	fDegreeOfLongitude :=,
	fDegreeOfLatitude := ,
	fReferenceMeridian := SEL( fb_GetTimeZoneInfo.tzID = eTimeZoneID_Daylight ,15,30),  (* Central European Time 15 Winter Timer / 30 Summer Time *)
	dCurrentDate := DT_TO_DATE(SYSTEMTIME_TO_Dt (prgSystemTime.structSystemTime)),
	todSunrise => todSunrise,
	todSunset => todSunset);
	
r_trig_on (clk := (FB_TimeSwitch_CH5.b_Output_On AND (DT_TO_TOD(systemtime_to_dt(prgSystemTime.structSystemTime))< (todSunrise +  T#1H))) OR (FB_TimeSwitch_CH5.b_Output_On AND m_UnderGroundMode));
r_trig_off (clk := NOT FB_TimeSwitch_CH5.b_Output_On);

RS_Outsidelight(	Set := r_trig_on.Q OR ((todSunset - T#2H) =  DT_TO_TOD(systemtime_to_dt(prgSystemTime.structSystemTime)) AND FB_TimeSwitch_CH5.b_Output_On AND NOT m_UnderGroundMode) OR b_Manual_On_CH5 ,
					Reset1 := r_trig_off.Q OR (((todSunrise +  T#1H)= DT_TO_TOD(systemtime_to_dt(prgSystemTime.structSystemTime))) AND NOT m_UnderGroundMode) OR b_Manual_Off_CH5,
					Q1 => b_LoadOn_CH5 );		
b_Out_CH5	:= NOT b_LoadOn_CH5;
	
FB_TimeSwitch_CH8(
	b_Enable:= b_Enable_Control_Coffee2_CH8, 
	b_StatusOn:= NOT b_Out_CH8, 
	structSystemTime:=prgSystemTime.structSystemTime , 
	byte_MoFr_Open_Hour:= byte_MoFr_Open_Hour , 
	byte_MoFr_Open_Minute:= byte_MoFr_Open_Minute, 
	byte_MoFr_Close_Hour:= byte_MoFr_Close_Hour , 
	byte_MoFr_Close_Minute:= byte_MoFr_Close_Minute, 
	byte_Sa_Open_Hour:= byte_Sa_Open_Hour, 
	byte_Sa_Open_Minute:= byte_Sa_Open_Minute , 
	byte_Sa_Close_Hour:= byte_Sa_Close_Hour , 
	byte_Sa_Close_Minute:= byte_Sa_Close_Minute, 
	byte_So_Open_Hour:= byte_So_Open_Hour, 
	byte_So_Open_Minute:= byte_So_Open_Minute, 
	byte_So_Close_Hour:= byte_So_Close_Hour, 
	byte_So_Close_Minute:= byte_So_Close_Minute, 
	real_Offset_Start:= real_Offset_Start_Coffee2_CH8 , 
	real_Offset_Stop:= real_Offset_Stop_Coffee2_CH8 , 
	b_On_Manual:= b_Manual_On_Coffee2_CH8, 
	b_Off_Manual:= b_Manual_Off_Coffee2_CH8, 
	b_Output_On=> b_LoadOn_CH8, 
	b_Error=> );
b_Out_CH8 := NOT FB_TimeSwitch_CH8.b_Output_On;

END_PROGRAM

// ---- FBs/EL3443_DPM/FB_EL3443_DPM.TcPOU
(*  This function block calls up the variant values supplied by the EL3443 terminal. The multiplexer channels of the terminal are queried by the use of selectors.
    Due to the multiplexing of the values in the variant values, reading the terminal information requires several PLC cycles.
    In contrast, values that can be retrieved via the process image are output cyclically. 
    
    To use the function block:
    ▪ the predefined PDO assignment "DPM" (DPM: Distributed Power Measurement) must be selected for the terminal under "Process data".
    
    ▪ Then the PLC data type (structure from the process data, MDP5001_341_93A85FAB) must be activated in the "PLC" tab of the terminal.
    
    ▪ After creating the data type, the PLC project must be rebuilt.
    
    ▪ Finally, the terminal must be linked to the function block on the "PLC" tab*)
    
FUNCTION_BLOCK FB_EL3443_DPM
VAR_INPUT
    bEnable : BOOL; //Enables the Variant values to be queried using the multiplexer functions of the block
    stEL3443_IO : MDP5001_341_7CD731EE;
				//MDP5001_341_93A85FAB; //External data type that can be generated within the terminal on the PLC tab
				// MDP5001_341_66E0DA41
END_VAr

VAR_OUTPUT
    stStatusTotal 	 : ST_EL3443_DPM_StatusTotal; //General cyclical process data
    stStatusPhase_L1 : ST_EL3443_DPM_StatusLx; //Phase L1 specific cyclical process data 
    stStatusPhase_L2 : ST_EL3443_DPM_StatusLx; //Phase L2 specific cyclical process data
    stStatusPhase_L3 : ST_EL3443_DPM_StatusLx; //Phase L3 specific cyclical process data
    stVariantValues  : ST_EL3443_DPM_VariantValues; //Variant Values (non-cyclical values). Due to the multiplexing of the values in the Variant Values, the reading of the terminal information requires several PLC cycles.
    
    pDpmData : POINTER TO ARRAY[1..20] OF UDINT;
    
    bError : BOOL; //Becomes TRUE as soon as an error situation occurs.
END_VAR

VAR
    {attribute 'no_copy'}
    astEL3443MuxReal_Ch1: ARRAY [0..nARRAYSIZEMUXREAL] OF ST_EL3443_DPM_MUX_REAL; //Structure for the (Real) Multiplexer Channel 1 contains the selector and a reference to the corresponding memory location
    {attribute 'no_copy'}
    astEL3443MuxReal_Ch2: ARRAY [0..nARRAYSIZEMUXREAL] OF ST_EL3443_DPM_MUX_REAL; //Structure for the (Real) Multiplexer Channel 2 contains the selector and a reference to the corresponding memory location
    {attribute 'no_copy'}
    astEL3443MuxReal_Ch3: ARRAY [0..nARRAYSIZEMUXREAL] OF ST_EL3443_DPM_MUX_REAL; //Structure for the (Real) Multiplexer Channel 3 contains the selector and a reference to the corresponding memory location
    {attribute 'no_copy'}
    stEL3443MuxUlint_Ch4: ARRAY [0..nARRAYSIZEMUXULINT] OF ST_EL3443_DPM_MUX_ULINT; //Structure for the (ULINT/LINT) multiplexer channel 4 contains the selector and a pointer to the corresponding memory location
    
    {attribute 'no_copy'}
    bInit : BOOL; //Flag to indicate the initialised state of the function block
    nMuxRealState : INT := 0; //Position der Multplexer-Abfragen (Channel 1-3 (REAL))
    nCounterNotRepliedMuxReal : INT; //Number of cycles in which the multiplexer has not responded
    nMuxUlintState : INT := 0; //Position der Multplexer-Abfragen (Channel 4 (ULINT))
    nCounterNotRepliedMuxUlint : INT; //Number of cycles in which the multiplexer has not responded
    
    {attribute 'no_copy'}
    nNumberOfSelectorsCh1 : UINT; //number of selectors in channel 1
    {attribute 'no_copy'}
    nNumberOfSelectorsCh2 : UINT; //number of selectors in channel 2
    {attribute 'no_copy'}
    nNumberOfSelectorsCh3 : UINT; //number of selectors in channel 3
    {attribute 'no_copy'}
    nNumberOfSelectorsCh4 : UINT; //number of selectors in channel 4      
END_VAR

VAR CONSTANT
    nARRAYSIZEMUXREAL : INT := 122; //Array size of the REAL multiplexer channel
    nARRAYSIZEMUXULINT : INT := 74; //Array size of the ULINT multiplexer channel
    nERROR_NOT_REPLIED : INT := 10; //Maximum number of cycles the multiplexer may use before the error output is set 
END_VAR

//The output bError is set if the block is enabled and one of the multiplexer channels does not respond
bError := bEnable AND (nCounterNotRepliedMuxUlint >= nERROR_NOT_REPLIED OR nCounterNotRepliedMuxReal >= nERROR_NOT_REPLIED) ;

IF bEnable THEN
      
    IF NOT bInit THEN
        bInit := TRUE;
        Initialize();
    END_IF
    
    //===================================================================================================================================
    // Multiplexer channels 1-3 (REAL)

    //comparison of the transmitting and receiving selectors 
    IF astEL3443MuxReal_Ch1[nMuxRealState].nSelector = stEL3443_IO.MDP5001_341_Input.MDP5001_341_Total_Variant_Value_In_Index_1_REAL AND
       astEL3443MuxReal_Ch2[nMuxRealState].nSelector = stEL3443_IO.MDP5001_341_Input.MDP5001_341_Total_Variant_Value_In_Index_2_REAL AND 
       astEL3443MuxReal_Ch3[nMuxRealState].nSelector = stEL3443_IO.MDP5001_341_Input.MDP5001_341_Total_Variant_Value_In_Index_3_REAL THEN
        												
    
        //assignment of the received values to the referenced references
        IF __ISVALIDREF(astEL3443MuxReal_Ch1[nMuxRealState].fValueRef) THEN
            astEL3443MuxReal_Ch1[nMuxRealState].fValueRef := stEL3443_IO.MDP5001_341_Input.MDP5001_341_Total_Variant_Value_In_Value_1_REAL;
        END_IF
        IF __ISVALIDREF(astEL3443MuxReal_Ch2[nMuxRealState].fValueRef) THEN
            astEL3443MuxReal_Ch2[nMuxRealState].fValueRef := stEL3443_IO.MDP5001_341_Input.MDP5001_341_Total_Variant_Value_In_Value_2_REAL;
        END_IF
        IF __ISVALIDREF(astEL3443MuxReal_Ch3[nMuxRealState].fValueRef) THEN
            astEL3443MuxReal_Ch3[nMuxRealState].fValueRef := stEL3443_IO.MDP5001_341_Input.MDP5001_341_Total_Variant_Value_In_Value_3_REAL;
        END_IF
       
       //selection of the new selector group
       nMuxRealState := nMuxRealState + 1;
     
       IF nMuxRealState > nARRAYSIZEMUXREAL THEN
         nMuxRealState := 0;  
       END_IF
       
       nCounterNotRepliedMuxReal := 0;
    ELSIF
        stEL3443_IO.MDP5001_341_Input.MDP5001_341_Total_Variant_Value_In_Index_1_REAL = E_EL3443_DPM_Phase.Error_INDEX_Not_Valid OR    
        stEL3443_IO.MDP5001_341_Input.MDP5001_341_Total_Variant_Value_In_Index_2_REAL = E_EL3443_DPM_Phase.Error_INDEX_Not_Valid OR 
        stEL3443_IO.MDP5001_341_Input.MDP5001_341_Total_Variant_Value_In_Index_3_REAL = E_EL3443_DPM_Phase.Error_INDEX_Not_Valid THEN
    
        nCounterNotRepliedMuxReal := MIN(nCounterNotRepliedMuxReal + 1,nERROR_NOT_REPLIED);
    ELSE
        nCounterNotRepliedMuxReal := MIN(nCounterNotRepliedMuxReal + 1,nERROR_NOT_REPLIED); 
    END_IF
       
    // transfer of the selectors to the process image 
    stEL3443_IO.MDP5001_341_Output.MDP5001_341_Total_Variant_Value_Out_Index_1_REAL := astEL3443MuxReal_Ch1[nMuxRealState].nSelector;
    stEL3443_IO.MDP5001_341_Output.MDP5001_341_Total_Variant_Value_Out_Index_2_REAL := astEL3443MuxReal_Ch2[nMuxRealState].nSelector;
    stEL3443_IO.MDP5001_341_Output.MDP5001_341_Total_Variant_Value_Out_Index_3_REAL := astEL3443MuxReal_Ch3[nMuxRealState].nSelector;
    
    //===================================================================================================================================
    // Multiplexer channels 4 (ULINT)
    
    //comparison of the transmitting and receiving selector
    IF stEL3443MuxUlint_Ch4[nMuxUlintState].nSelector = stEL3443_IO.MDP5001_341_Input.MDP5001_341_Total_Variant_Value_In_Index_4_ULINT THEN
        
        //assigns the received values to the assigned pointer address.
        IF stEL3443MuxUlint_Ch4[nMuxUlintState].nValueRef <> 0 THEN
            stEL3443MuxUlint_Ch4[nMuxUlintState].nValueRef^ := stEL3443_IO.MDP5001_341_Input.MDP5001_341_Total_Variant_Value_In_Value_4_ULINT;
        END_IF
        
    //selection of the new selector group
       nMuxUlintState := nMuxUlintState + 1;
     
       IF nMuxUlintState > nARRAYSIZEMUXULINT THEN
         nMuxUlintState := 0;  
       END_IF
       
       nCounterNotRepliedMuxUlint := 0;
    ELSIF stEL3443_IO.MDP5001_341_Input.MDP5001_341_Total_Variant_Value_In_Index_4_ULINT = E_EL3443_DPM_Phase.Error_INDEX_Not_Valid THEN
    
        nCounterNotRepliedMuxUlint := MIN(nCounterNotRepliedMuxUlint + 1, nERROR_NOT_REPLIED);
    ELSE
        nCounterNotRepliedMuxUlint := MIN(nCounterNotRepliedMuxUlint + 1, nERROR_NOT_REPLIED);  
    END_IF
    
    // transfer of the selectors to the process image
    stEL3443_IO.MDP5001_341_Output.MDP5001_341_Total_Variant_Value_Out_Index_4_ULINT := stEL3443MuxUlint_Ch4[nMuxUlintState].nSelector;
END_IF

//===================================================================================================================================
// Update the cyclic outputs

// Set pointer address to transmit DPM communication information
pDpmData := ADR(stEL3443_IO.MDP5001_341_Input.MDP5001_341_DPM_Data_Data_1);

// Transfer of process data to PLC common data types. Status total.
stStatusTotal.bStatus_System_State :=                       stEL3443_IO.MDP5001_341_Input.MDP5001_341_Total_Status_System_State;
stStatusTotal.bStatus_Grid_Direction :=                     stEL3443_IO.MDP5001_341_Input.MDP5001_341_Total_Status_Grid_Direction;
stStatusTotal.bStatus_Frequency_Guard_Warning :=            stEL3443_IO.MDP5001_341_Input.MDP5001_341_Total_Status_Frequency_Guard_Warning;
stStatusTotal.bStatus_Frequency_Guard_Error :=              stEL3443_IO.MDP5001_341_Input.MDP5001_341_Total_Status_Frequency_Guard_Error;
stStatusTotal.bStatus_Neutral_Current_Guard_Warning :=      stEL3443_IO.MDP5001_341_Input.MDP5001_341_Total_Status_Neutral_Current_Guard_Warning;
stStatusTotal.bStatus_Neutral_Current_Guard_Error :=        stEL3443_IO.MDP5001_341_Input.MDP5001_341_Total_Status_Neutral_Current_Guard_Error;
stStatusTotal.bStatus_Active_Power_Guard_Warning :=         stEL3443_IO.MDP5001_341_Input.MDP5001_341_Total_Status_Active_Power_Guard_Warning;    
stStatusTotal.bStatus_Active_Power_Guard_Error :=           stEL3443_IO.MDP5001_341_Input.MDP5001_341_Total_Status_Active_Power_Guard_Error;
stStatusTotal.bStatus_Apparent_Power_Guard_Warning :=       stEL3443_IO.MDP5001_341_Input.MDP5001_341_Total_Status_Apparent_Power_Guard_Warning;
stStatusTotal.bStatus_Apparent_Power_Guard_Error :=         stEL3443_IO.MDP5001_341_Input.MDP5001_341_Total_Status_Apparent_Power_Guard_Error; 
stStatusTotal.bStatus_Power_Quality_Guard_Warning :=        stEL3443_IO.MDP5001_341_Input.MDP5001_341_Total_Status_Power_Quality_Guard_Warning; 
stStatusTotal.bStatus_Power_Quality_Guard_Error :=          stEL3443_IO.MDP5001_341_Input.MDP5001_341_Total_Status_Power_Quality_Guard_Error; 
stStatusTotal.bStatus_TxPDO_State :=                        stEL3443_IO.MDP5001_341_Input.MDP5001_341_Total_Status_TxPDO_State; 
stStatusTotal.bStatus_TxPDO_Toggle :=                       stEL3443_IO.MDP5001_341_Input.MDP5001_341_Total_Status_TxPDO_Toggle; 
stStatusTotal.fStatus_Power_Quality_Factor :=               stEL3443_IO.MDP5001_341_Input.MDP5001_341_Total_Status_Power_Quality_Factor; 

//Transfer of process data to PLC common data types. Status phase L1.
stStatusPhase_L1.bStatus_Voltage_Sign_Bit  :=               stEL3443_IO.MDP5001_341_Input.MDP5001_341_L1_Status_Voltage_Sign_Bit;
stStatusPhase_L1.bStatus_Overvoltage  :=                    stEL3443_IO.MDP5001_341_Input.MDP5001_341_L1_Status_Overvoltage;
stStatusPhase_L1.bStatus_Overcurrent  :=                    stEL3443_IO.MDP5001_341_Input.MDP5001_341_L1_Status_Overcurrent;
stStatusPhase_L1.bStatus_Inaccurate_Voltage  :=             stEL3443_IO.MDP5001_341_Input.MDP5001_341_L1_Status_Inaccurate_Voltage;
stStatusPhase_L1.bStatus_Inaccurate_Current  :=             stEL3443_IO.MDP5001_341_Input.MDP5001_341_L1_Status_Inaccurate_Current;
stStatusPhase_L1.bStatus_Voltage_Guard_Warning  :=          stEL3443_IO.MDP5001_341_Input.MDP5001_341_L1_Status_Voltage_Guard_Warning;
stStatusPhase_L1.bStatus_Voltage_Guard_Error  :=            stEL3443_IO.MDP5001_341_Input.MDP5001_341_L1_Status_Voltage_Guard_Error;
stStatusPhase_L1.bStatus_Current_Guard_Warning  :=          stEL3443_IO.MDP5001_341_Input.MDP5001_341_L1_Status_Current_Guard_Warning;
stStatusPhase_L1.bStatus_Current_Guard_Error  :=            stEL3443_IO.MDP5001_341_Input.MDP5001_341_L1_Status_Current_Guard_Error;
stStatusPhase_L1.bStatus_TxPDO_Toggle  :=                   stEL3443_IO.MDP5001_341_Input.MDP5001_341_L1_Status_TxPDO_Toggle;

//Transfer of process data to PLC common data types. Status phase L2.
stStatusPhase_L2.bStatus_Voltage_Sign_Bit  :=               stEL3443_IO.MDP5001_341_Input.MDP5001_341_L2_Status_Voltage_Sign_Bit;
stStatusPhase_L2.bStatus_Overvoltage  :=                    stEL3443_IO.MDP5001_341_Input.MDP5001_341_L2_Status_Overvoltage;
stStatusPhase_L2.bStatus_Overcurrent  :=                    stEL3443_IO.MDP5001_341_Input.MDP5001_341_L2_Status_Overcurrent;        
stStatusPhase_L2.bStatus_Inaccurate_Voltage  :=             stEL3443_IO.MDP5001_341_Input.MDP5001_341_L2_Status_Inaccurate_Voltage;		
stStatusPhase_L2.bStatus_Inaccurate_Current  :=             stEL3443_IO.MDP5001_341_Input.MDP5001_341_L2_Status_Inaccurate_Current;		
stStatusPhase_L2.bStatus_Voltage_Guard_Warning  :=          stEL3443_IO.MDP5001_341_Input.MDP5001_341_L2_Status_Voltage_Guard_Warning;		
stStatusPhase_L2.bStatus_Voltage_Guard_Error  :=            stEL3443_IO.MDP5001_341_Input.MDP5001_341_L2_Status_Voltage_Guard_Error;		
stStatusPhase_L2.bStatus_Current_Guard_Warning  :=          stEL3443_IO.MDP5001_341_Input.MDP5001_341_L2_Status_Current_Guard_Warning;		
stStatusPhase_L2.bStatus_Current_Guard_Error  :=            stEL3443_IO.MDP5001_341_Input.MDP5001_341_L2_Status_Current_Guard_Error;		
stStatusPhase_L2.bStatus_TxPDO_Toggle  :=                   stEL3443_IO.MDP5001_341_Input.MDP5001_341_L2_Status_TxPDO_Toggle;		
		
//Transfer of process data to PLC common data types. Status phase L3.		
stStatusPhase_L3.bStatus_Voltage_Sign_Bit  :=               stEL3443_IO.MDP5001_341_Input.MDP5001_341_L3_Status_Voltage_Sign_Bit;		
stStatusPhase_L3.bStatus_Overvoltage  :=                    stEL3443_IO.MDP5001_341_Input.MDP5001_341_L3_Status_Overvoltage;                                             
stStatusPhase_L3.bStatus_Overcurrent  :=                    stEL3443_IO.MDP5001_341_Input.MDP5001_341_L3_Status_Overcurrent;
stStatusPhase_L3.bStatus_Inaccurate_Voltage  :=             stEL3443_IO.MDP5001_341_Input.MDP5001_341_L3_Status_Inaccurate_Voltage;
stStatusPhase_L3.bStatus_Inaccurate_Current  :=             stEL3443_IO.MDP5001_341_Input.MDP5001_341_L3_Status_Inaccurate_Current;
stStatusPhase_L3.bStatus_Voltage_Guard_Warning  :=          stEL3443_IO.MDP5001_341_Input.MDP5001_341_L3_Status_Voltage_Guard_Warning;
stStatusPhase_L3.bStatus_Voltage_Guard_Error  :=            stEL3443_IO.MDP5001_341_Input.MDP5001_341_L3_Status_Voltage_Guard_Error;
stStatusPhase_L3.bStatus_Current_Guard_Warning  :=          stEL3443_IO.MDP5001_341_Input.MDP5001_341_L3_Status_Current_Guard_Warning;
stStatusPhase_L3.bStatus_Current_Guard_Error  :=            stEL3443_IO.MDP5001_341_Input.MDP5001_341_L3_Status_Current_Guard_Error;
stStatusPhase_L3.bStatus_TxPDO_Toggle  :=                   stEL3443_IO.MDP5001_341_Input.MDP5001_341_L3_Status_TxPDO_Toggle;

(* This method initializes the lookup table and establishes a connection between selector index and variable by references. *)
METHOD PRIVATE Initialize : HRESULT
VAR
    nPhase : INT; // Three-phase
    stEL3443MuxReal : REFERENCE TO ARRAY [0..nARRAYSIZEMUXREAL] OF ST_EL3443_DPM_MUX_REAL;
    nNumberOfSelector : REFERENCE TO UINT;
    nOFFSET : UINT;
    i : UINT;
END_VAR
// - The process data of phases L1, L2 and L3 are distributed to the three REAL multiplexers. (Channel1 = L1, Channel2 = L2 ...)
// - The ULINT multiplexer is initialized with data from all three phases.
FOR nPhase := 1 TO 3 DO
    
    // Selection of the structures, selector counters and offset based on the phase
    CASE nPhase OF
    1: // Phase L1
       stEL3443MuxReal REF= astEL3443MuxReal_Ch1;
       nNumberOfSelector REF= nNumberOfSelectorsCh1;
       nOFFSET := E_EL3443_DPM_Phase.nPhaseL1_OFFSET;  
    2: // Phase L2 
       stEL3443MuxReal REF= astEL3443MuxReal_Ch2;
       nNumberOfSelector REF= nNumberOfSelectorsCh2;
       nOFFSET := E_EL3443_DPM_Phase.nPhaseL2_OFFSET; 
    3: // Phase L3 
       stEL3443MuxReal REF= astEL3443MuxReal_Ch3;
       nNumberOfSelector REF= nNumberOfSelectorsCh3;
       nOFFSET := E_EL3443_DPM_Phase.nPhaseL3_OFFSET;
    ELSE
       EXIT;   
	END_CASE
    
    // Initializing the REAL multiplexers on channels 1 to 3
    InitSelectorReal(stEL3443MuxReal, nNumberOfSelector, stVariantValues.astLx[nPhase].fU_RMS,         nOFFSET, E_EL3443_DPM_Phase.U_RMS         );
    InitSelectorReal(stEL3443MuxReal, nNumberOfSelector, stVariantValues.astLx[nPhase].fU_peak,        nOFFSET, E_EL3443_DPM_Phase.U_peak        );
    InitSelectorReal(stEL3443MuxReal, nNumberOfSelector, stVariantValues.astLx[nPhase].fU_RMS_Minimum, nOFFSET, E_EL3443_DPM_Phase.U_RMS_Minimum);
    InitSelectorReal(stEL3443MuxReal, nNumberOfSelector, stVariantValues.astLx[nPhase].fU_RMS_Maximum, nOFFSET, E_EL3443_DPM_Phase.U_RMS_Maximum);
    InitSelectorReal(stEL3443MuxReal, nNumberOfSelector, stVariantValues.astLx[nPhase].fULL,           nOFFSET, E_EL3443_DPM_Phase.ULL          );
    InitSelectorReal(stEL3443MuxReal, nNumberOfSelector, stVariantValues.astLx[nPhase].fI_RMS,         nOFFSET, E_EL3443_DPM_Phase.I_RMS        );
    InitSelectorReal(stEL3443MuxReal, nNumberOfSelector, stVariantValues.astLx[nPhase].fI_peak,        nOFFSET, E_EL3443_DPM_Phase.I_peak       ); 
    InitSelectorReal(stEL3443MuxReal, nNumberOfSelector, stVariantValues.astLx[nPhase].fI_RMS_Minimum, nOFFSET, E_EL3443_DPM_Phase.I_RMS_Minimum );
    InitSelectorReal(stEL3443MuxReal, nNumberOfSelector, stVariantValues.astLx[nPhase].fI_RMS_Maximum, nOFFSET, E_EL3443_DPM_Phase.I_RMS_Maximum );
    InitSelectorReal(stEL3443MuxReal, nNumberOfSelector, stVariantValues.astLx[nPhase].fFrequency,     nOFFSET, E_EL3443_DPM_Phase.Frequency     );
    InitSelectorReal(stEL3443MuxReal, nNumberOfSelector, stVariantValues.astLx[nPhase].fPhi,           nOFFSET, E_EL3443_DPM_Phase.Phi,          );
    InitSelectorReal(stEL3443MuxReal, nNumberOfSelector, stVariantValues.astLx[nPhase].fCOS_phi,       nOFFSET, E_EL3443_DPM_Phase.Cos_phi       );
    InitSelectorReal(stEL3443MuxReal, nNumberOfSelector, stVariantValues.astLx[nPhase].fPower_Factor,  nOFFSET, E_EL3443_DPM_Phase.Power_Factor  );
    InitSelectorReal(stEL3443MuxReal, nNumberOfSelector, stVariantValues.astLx[nPhase].fP,             nOFFSET, E_EL3443_DPM_Phase.P             );
    InitSelectorReal(stEL3443MuxReal, nNumberOfSelector, stVariantValues.astLx[nPhase].fPavg,          nOFFSET, E_EL3443_DPM_Phase.Pavg          );
    InitSelectorReal(stEL3443MuxReal, nNumberOfSelector, stVariantValues.astLx[nPhase].fPmin,          nOFFSET, E_EL3443_DPM_Phase.Pmin          );
    InitSelectorReal(stEL3443MuxReal, nNumberOfSelector, stVariantValues.astLx[nPhase].fPmax,          nOFFSET, E_EL3443_DPM_Phase.Pmax          );
    InitSelectorReal(stEL3443MuxReal, nNumberOfSelector, stVariantValues.astLx[nPhase].fS,             nOFFSET, E_EL3443_DPM_Phase.S_            );
    InitSelectorReal(stEL3443MuxReal, nNumberOfSelector, stVariantValues.astLx[nPhase].fSavg,          nOFFSET, E_EL3443_DPM_Phase.Savg          );
    InitSelectorReal(stEL3443MuxReal, nNumberOfSelector, stVariantValues.astLx[nPhase].fSmin,          nOFFSET, E_EL3443_DPM_Phase.Smin          );
    InitSelectorReal(stEL3443MuxReal, nNumberOfSelector, stVariantValues.astLx[nPhase].fSmax,          nOFFSET, E_EL3443_DPM_Phase.Smax          );
    InitSelectorReal(stEL3443MuxReal, nNumberOfSelector, stVariantValues.astLx[nPhase].fQ,             nOFFSET, E_EL3443_DPM_Phase.Q             );
    InitSelectorReal(stEL3443MuxReal, nNumberOfSelector, stVariantValues.astLx[nPhase].fQavg,          nOFFSET, E_EL3443_DPM_Phase.Qavg          );
    InitSelectorReal(stEL3443MuxReal, nNumberOfSelector, stVariantValues.astLx[nPhase].fQmin,          nOFFSET, E_EL3443_DPM_Phase.Qmin          );
    InitSelectorReal(stEL3443MuxReal, nNumberOfSelector, stVariantValues.astLx[nPhase].fQmax,          nOFFSET, E_EL3443_DPM_Phase.Qmax          );
    InitSelectorReal(stEL3443MuxReal, nNumberOfSelector, stVariantValues.astLx[nPhase].fTHD_U,         nOFFSET, E_EL3443_DPM_Phase.THD_U         );     
    InitSelectorReal(stEL3443MuxReal, nNumberOfSelector, stVariantValues.astLx[nPhase].fRMS_fund_U,    nOFFSET, E_EL3443_DPM_Phase.RMS_fund_U    );
    InitSelectorReal(stEL3443MuxReal, nNumberOfSelector, stVariantValues.astLx[nPhase].fF_Ref_U,       nOFFSET, E_EL3443_DPM_Phase.F_Ref_U       );
    InitSelectorReal(stEL3443MuxReal, nNumberOfSelector, stVariantValues.astLx[nPhase].fTHD_I,         nOFFSET, E_EL3443_DPM_Phase.THD_I        );
    InitSelectorReal(stEL3443MuxReal, nNumberOfSelector, stVariantValues.astLx[nPhase].fTDD_I,         nOFFSET, E_EL3443_DPM_Phase.TDD_I        );
    InitSelectorReal(stEL3443MuxReal, nNumberOfSelector, stVariantValues.astLx[nPhase].fRMS_fund_I,    nOFFSET, E_EL3443_DPM_Phase.RMS_fund_I   );
    InitSelectorReal(stEL3443MuxReal, nNumberOfSelector, stVariantValues.astLx[nPhase].fF_Ref_I,       nOFFSET, E_EL3443_DPM_Phase.F_Ref_I      );
    
    // Initializing the Real Arrays on channel 1 to 3
    FOR i := 0 TO 41 DO
        InitSelectorReal(stEL3443MuxReal, nNumberOfSelector, stVariantValues.astLx[nPhase].fHarmonics_U[i], nOFFSET  + i, E_EL3443_DPM_Phase.Harmonics_U);
    END_FOR
    FOR i := 0 TO 41 DO
        InitSelectorReal(stEL3443MuxReal, nNumberOfSelector, stVariantValues.astLx[nPhase].fHarmonics_I[i], nOFFSET  + i, E_EL3443_DPM_Phase.Harmonics_I);   
    END_FOR

    // Initializing the ULINT multiplexer on channel 4
    InitSelectorUlint(stEL3443MuxUlint_Ch4, nNumberOfSelectorsCh4, stVariantValues.astLx[nPhase].nU_Last_Zero_Cross, nOFFSET, E_EL3443_DPM_Phase.U_Last_Zero_Cross	);
    InitSelectorUlint(stEL3443MuxUlint_Ch4, nNumberOfSelectorsCh4, stVariantValues.astLx[nPhase].nEP,                nOFFSET, E_EL3443_DPM_Phase.EP               	);
    InitSelectorUlint(stEL3443MuxUlint_Ch4, nNumberOfSelectorsCh4, stVariantValues.astLx[nPhase].nEP_pos,            nOFFSET, E_EL3443_DPM_Phase.EP_pos           	);
    InitSelectorUlint(stEL3443MuxUlint_Ch4, nNumberOfSelectorsCh4, stVariantValues.astLx[nPhase].nEP_neg,            nOFFSET, E_EL3443_DPM_Phase.EP_neg          	);
    InitSelectorUlint(stEL3443MuxUlint_Ch4, nNumberOfSelectorsCh4, stVariantValues.astLx[nPhase].nEP_interval,    	 nOFFSET, E_EL3443_DPM_Phase.EP_interval    	);
    InitSelectorUlint(stEL3443MuxUlint_Ch4, nNumberOfSelectorsCh4, stVariantValues.astLx[nPhase].nEP_pos_interval,	 nOFFSET, E_EL3443_DPM_Phase.EP_pos_interval	);
    InitSelectorUlint(stEL3443MuxUlint_Ch4, nNumberOfSelectorsCh4, stVariantValues.astLx[nPhase].nEP_neg_interval,	 nOFFSET, E_EL3443_DPM_Phase.EP_neg_interval	);
	InitSelectorUlint(stEL3443MuxUlint_Ch4, nNumberOfSelectorsCh4, stVariantValues.astLx[nPhase].nES,                nOFFSET, E_EL3443_DPM_Phase.ES               	);
    InitSelectorUlint(stEL3443MuxUlint_Ch4, nNumberOfSelectorsCh4, stVariantValues.astLx[nPhase].nES_pos,            nOFFSET, E_EL3443_DPM_Phase.ES_pos           	);
    InitSelectorUlint(stEL3443MuxUlint_Ch4, nNumberOfSelectorsCh4, stVariantValues.astLx[nPhase].nES_neg,            nOFFSET, E_EL3443_DPM_Phase.ES_neg          	);
    InitSelectorUlint(stEL3443MuxUlint_Ch4, nNumberOfSelectorsCh4, stVariantValues.astLx[nPhase].nES_interval,    	 nOFFSET, E_EL3443_DPM_Phase.ES_interval    	);
    InitSelectorUlint(stEL3443MuxUlint_Ch4, nNumberOfSelectorsCh4, stVariantValues.astLx[nPhase].nES_pos_interval,	 nOFFSET, E_EL3443_DPM_Phase.ES_pos_interval	);
    InitSelectorUlint(stEL3443MuxUlint_Ch4, nNumberOfSelectorsCh4, stVariantValues.astLx[nPhase].nES_neg_interval,	 nOFFSET, E_EL3443_DPM_Phase.ES_neg_interval	);
	InitSelectorUlint(stEL3443MuxUlint_Ch4, nNumberOfSelectorsCh4, stVariantValues.astLx[nPhase].nEQ,                nOFFSET, E_EL3443_DPM_Phase.EQ_              	);
    InitSelectorUlint(stEL3443MuxUlint_Ch4, nNumberOfSelectorsCh4, stVariantValues.astLx[nPhase].nEQ_pos,            nOFFSET, E_EL3443_DPM_Phase.EQ_pos           	);
    InitSelectorUlint(stEL3443MuxUlint_Ch4, nNumberOfSelectorsCh4, stVariantValues.astLx[nPhase].nEQ_neg,            nOFFSET, E_EL3443_DPM_Phase.EQ_neg           	);
    InitSelectorUlint(stEL3443MuxUlint_Ch4, nNumberOfSelectorsCh4, stVariantValues.astLx[nPhase].nEQ_interval,    	 nOFFSET, E_EL3443_DPM_Phase.EQ_interval    	);
    InitSelectorUlint(stEL3443MuxUlint_Ch4, nNumberOfSelectorsCh4, stVariantValues.astLx[nPhase].nEQ_pos_interval,	 nOFFSET, E_EL3443_DPM_Phase.EQ_pos_interval	);
    InitSelectorUlint(stEL3443MuxUlint_Ch4, nNumberOfSelectorsCh4, stVariantValues.astLx[nPhase].nEQ_neg_interval,	 nOFFSET, E_EL3443_DPM_Phase.EQ_neg_interval	);        
END_FOR

// All data that is not assigned to a phase is appended to channels 1 to 4. 

// Real values for multiplexer channel 1   
InitSelectorReal(astEL3443MuxReal_Ch1, nNumberOfSelectorsCh1, stVariantValues.stTotal.fIn_RMS,         E_EL3443_DPM_Total.nTotal_OFFSET, E_EL3443_DPM_Total.In_RMS        );
InitSelectorReal(astEL3443MuxReal_Ch1, nNumberOfSelectorsCh1, stVariantValues.stTotal.fPower_Factor,   E_EL3443_DPM_Total.nTotal_OFFSET, E_EL3443_DPM_Total.Power_Factor  );
InitSelectorReal(astEL3443MuxReal_Ch1, nNumberOfSelectorsCh1, stVariantValues.stTotal.fPtot,           E_EL3443_DPM_Total.nTotal_OFFSET, E_EL3443_DPM_Total.Ptot          );
InitSelectorReal(astEL3443MuxReal_Ch1, nNumberOfSelectorsCh1, stVariantValues.stTotal.fPtotavg,        E_EL3443_DPM_Total.nTotal_OFFSET, E_EL3443_DPM_Total.Ptotavg       );
InitSelectorReal(astEL3443MuxReal_Ch1, nNumberOfSelectorsCh1, stVariantValues.stTotal.fPtotmin,        E_EL3443_DPM_Total.nTotal_OFFSET, E_EL3443_DPM_Total.Ptotmin       );
InitSelectorReal(astEL3443MuxReal_Ch1, nNumberOfSelectorsCh1, stVariantValues.stTotal.fPtotmax,        E_EL3443_DPM_Total.nTotal_OFFSET, E_EL3443_DPM_Total.Ptotmax       );
InitSelectorReal(astEL3443MuxReal_Ch1, nNumberOfSelectorsCh1, stVariantValues.stTotal.fStot,           E_EL3443_DPM_Total.nTotal_OFFSET, E_EL3443_DPM_Total.Stot          );

// Real values for multiplexer channel 2
InitSelectorReal(astEL3443MuxReal_Ch2, nNumberOfSelectorsCh2, stVariantValues.stTotal.fStotavg,   E_EL3443_DPM_Total.nTotal_OFFSET, E_EL3443_DPM_Total.Stotavg);                                                                                                                        
InitSelectorReal(astEL3443MuxReal_Ch2, nNumberOfSelectorsCh2, stVariantValues.stTotal.fStotmin,   E_EL3443_DPM_Total.nTotal_OFFSET, E_EL3443_DPM_Total.Stotmin);
InitSelectorReal(astEL3443MuxReal_Ch2, nNumberOfSelectorsCh2, stVariantValues.stTotal.fStotmax,   E_EL3443_DPM_Total.nTotal_OFFSET, E_EL3443_DPM_Total.Stotmax);
InitSelectorReal(astEL3443MuxReal_Ch2, nNumberOfSelectorsCh2, stVariantValues.stTotal.fQtot,      E_EL3443_DPM_Total.nTotal_OFFSET, E_EL3443_DPM_Total.Qtot   );
InitSelectorReal(astEL3443MuxReal_Ch2, nNumberOfSelectorsCh2, stVariantValues.stTotal.fQtotavg,   E_EL3443_DPM_Total.nTotal_OFFSET, E_EL3443_DPM_Total.Qtotavg);
InitSelectorReal(astEL3443MuxReal_Ch2, nNumberOfSelectorsCh2, stVariantValues.stTotal.fQtotmin,   E_EL3443_DPM_Total.nTotal_OFFSET, E_EL3443_DPM_Total.Qtotmin);
InitSelectorReal(astEL3443MuxReal_Ch2, nNumberOfSelectorsCh2, stVariantValues.stTotal.fQtotmax,   E_EL3443_DPM_Total.nTotal_OFFSET, E_EL3443_DPM_Total.Qtotmax);

//Real values for multiplexer channel 3
InitSelectorReal(astEL3443MuxReal_Ch3, nNumberOfSelectorsCh3, stVariantValues.stTotal.fPhiL1L2,   E_EL3443_DPM_Total.nTotal_OFFSET, E_EL3443_DPM_Total.PhiL1L2  );
InitSelectorReal(astEL3443MuxReal_Ch3, nNumberOfSelectorsCh3, stVariantValues.stTotal.fPhiL1L3,   E_EL3443_DPM_Total.nTotal_OFFSET, E_EL3443_DPM_Total.PhiL1L3  );
InitSelectorReal(astEL3443MuxReal_Ch3, nNumberOfSelectorsCh3, stVariantValues.stTotal.fUnbalance, E_EL3443_DPM_Total.nTotal_OFFSET, E_EL3443_DPM_Total.Unbalance);
InitSelectorReal(astEL3443MuxReal_Ch3, nNumberOfSelectorsCh3, stVariantValues.stTotal.fPQF,       E_EL3443_DPM_Total.nTotal_OFFSET, E_EL3443_DPM_Total.PQF      );
InitSelectorReal(astEL3443MuxReal_Ch3, nNumberOfSelectorsCh3, stVariantValues.stTotal.fPQF_Avg,   E_EL3443_DPM_Total.nTotal_OFFSET, E_EL3443_DPM_Total.PQF_Avg  );
InitSelectorReal(astEL3443MuxReal_Ch3, nNumberOfSelectorsCh3, stVariantValues.stTotal.fPQF_Min,   E_EL3443_DPM_Total.nTotal_OFFSET, E_EL3443_DPM_Total.PQF_MIN  );
InitSelectorReal(astEL3443MuxReal_Ch3, nNumberOfSelectorsCh3, stVariantValues.stTotal.fPQF_Max,   E_EL3443_DPM_Total.nTotal_OFFSET, E_EL3443_DPM_Total.PQF_MAX);


// Ulint values for multiplexer channel 4
InitSelectorUlint(stEL3443MuxUlint_Ch4, nNumberOfSelectorsCh4, stVariantValues.stTotal.nEptot,                    E_EL3443_DPM_Total.nTotal_OFFSET, E_EL3443_DPM_Total.Eptot         	);
InitSelectorUlint(stEL3443MuxUlint_Ch4, nNumberOfSelectorsCh4, stVariantValues.stTotal.nEPtot_pos,                E_EL3443_DPM_Total.nTotal_OFFSET, E_EL3443_DPM_Total.EPtot_pos        );
InitSelectorUlint(stEL3443MuxUlint_Ch4, nNumberOfSelectorsCh4, stVariantValues.stTotal.nEPtot_neg,                E_EL3443_DPM_Total.nTotal_OFFSET, E_EL3443_DPM_Total.EPtot_neg        );
InitSelectorUlint(stEL3443MuxUlint_Ch4, nNumberOfSelectorsCh4, stVariantValues.stTotal.nEptot_interval,          E_EL3443_DPM_Total.nTotal_OFFSET, E_EL3443_DPM_Total.Eptot_interval    );
InitSelectorUlint(stEL3443MuxUlint_Ch4, nNumberOfSelectorsCh4, stVariantValues.stTotal.nEPtot_pos_interval,      E_EL3443_DPM_Total.nTotal_OFFSET, E_EL3443_DPM_Total.EPtot_pos_interval);
InitSelectorUlint(stEL3443MuxUlint_Ch4, nNumberOfSelectorsCh4, stVariantValues.stTotal.nEPtot_neg_interval,      E_EL3443_DPM_Total.nTotal_OFFSET, E_EL3443_DPM_Total.EPtot_neg_interval);
InitSelectorUlint(stEL3443MuxUlint_Ch4, nNumberOfSelectorsCh4, stVariantValues.stTotal.nEStot,                    E_EL3443_DPM_Total.nTotal_OFFSET, E_EL3443_DPM_Total.EStot            );
InitSelectorUlint(stEL3443MuxUlint_Ch4, nNumberOfSelectorsCh4, stVariantValues.stTotal.nEStot_pos,                E_EL3443_DPM_Total.nTotal_OFFSET, E_EL3443_DPM_Total.EStot_pos        );
InitSelectorUlint(stEL3443MuxUlint_Ch4, nNumberOfSelectorsCh4, stVariantValues.stTotal.nEStot_neg,                E_EL3443_DPM_Total.nTotal_OFFSET, E_EL3443_DPM_Total.EStot_neg        );
InitSelectorUlint(stEL3443MuxUlint_Ch4, nNumberOfSelectorsCh4, stVariantValues.stTotal.nEStot_interval,          E_EL3443_DPM_Total.nTotal_OFFSET, E_EL3443_DPM_Total.EStot_interval    );
InitSelectorUlint(stEL3443MuxUlint_Ch4, nNumberOfSelectorsCh4, stVariantValues.stTotal.nEStot_pos_interval,      E_EL3443_DPM_Total.nTotal_OFFSET, E_EL3443_DPM_Total.EStot_pos_interval);
InitSelectorUlint(stEL3443MuxUlint_Ch4, nNumberOfSelectorsCh4, stVariantValues.stTotal.nEStot_neg_interval,      E_EL3443_DPM_Total.nTotal_OFFSET, E_EL3443_DPM_Total.EStot_neg_interval);
InitSelectorUlint(stEL3443MuxUlint_Ch4, nNumberOfSelectorsCh4, stVariantValues.stTotal.nEQtot,                    E_EL3443_DPM_Total.nTotal_OFFSET, E_EL3443_DPM_Total.EQtot            );
InitSelectorUlint(stEL3443MuxUlint_Ch4, nNumberOfSelectorsCh4, stVariantValues.stTotal.nEQtot_pos,                E_EL3443_DPM_Total.nTotal_OFFSET, E_EL3443_DPM_Total.EQtot_pos        );
InitSelectorUlint(stEL3443MuxUlint_Ch4, nNumberOfSelectorsCh4, stVariantValues.stTotal.nEQtot_neg,                E_EL3443_DPM_Total.nTotal_OFFSET, E_EL3443_DPM_Total.EQtot_neg        );
InitSelectorUlint(stEL3443MuxUlint_Ch4, nNumberOfSelectorsCh4, stVariantValues.stTotal.nEQtot_interval,          E_EL3443_DPM_Total.nTotal_OFFSET, E_EL3443_DPM_Total.EQtot_interval    );
InitSelectorUlint(stEL3443MuxUlint_Ch4, nNumberOfSelectorsCh4, stVariantValues.stTotal.nEQtot_pos_interval,      E_EL3443_DPM_Total.nTotal_OFFSET, E_EL3443_DPM_Total.EQtot_pos_interval);
InitSelectorUlint(stEL3443MuxUlint_Ch4, nNumberOfSelectorsCh4, stVariantValues.stTotal.nEQtot_neg_interval,      E_EL3443_DPM_Total.nTotal_OFFSET, E_EL3443_DPM_Total.EQtot_neg_interval);
END_METHOD

(*This method calculates the selector based on the offset and the base selector and sets the corresponding reference*)
METHOD PRIVATE InitSelectorReal : HRESULT
VAR_IN_OUT
    stEL3443MuxReal : ARRAY [0..nARRAYSIZEMUXREAL] OF ST_EL3443_DPM_MUX_REAL;
    nNumberOfSelectors : UINT;    
    fValue : REAL;  
END_VAR
VAR_INPUT
    nOFFSET : UINT;
    nSelector : UINT;
END_VAR
    stEL3443MuxReal[nNumberOfSelectors].nSelector := nSelector + nOFFSET; //Basis Selector + Channel(Phase) Offset
    stEL3443MuxReal[nNumberOfSelectors].fValueRef REF= fValue; //Set reference to create a link between selector and output value
    nNumberOfSelectors := nNumberOfSelectors + 1;
END_METHOD

(*This method calculates the selector based on the offset and the base selector and sets the corresponding pointer address*)
METHOD PRIVATE InitSelectorUlint : HRESULT
VAR_IN_OUT
    stEL3443MuxUlint : ARRAY [0..nARRAYSIZEMUXULINT] OF ST_EL3443_DPM_MUX_ULINT;
    nNumberOfSelectors : UINT;  
END_VAR
VAR_INPUT
    nValue : ANY_INT;
    nOFFSET : UINT;
    nSelector : UINT;
END_VAR
    stEL3443MuxUlint[nNumberOfSelectors].nSelector := nSelector + nOFFSET; //Basis Selector + Channel(Phase) Offset
    stEL3443MuxUlint[nNumberOfSelectors].nValueRef := nValue.pValue; //Set reference to create a link between selector and output value
    nNumberOfSelectors := nNumberOfSelectors + 1;
END_METHOD

END_FUNCTION_BLOCK

// ---- FBs/FB_CoE_EL3446.TcPOU
FUNCTION_BLOCK FB_CoE_EL3446
VAR_INPUT
	m_start: BOOL;
	nSlaveAddr	:UINT;
	uiVoltagePhaseSelector_CH1		: UINT;											//Voltage Phase Selector 1/2/3 for Channel 1
	uiVoltagePhaseSelector_CH2		: UINT;											//Voltage Phase Selector 1/2/3 for Channel 2
	uiVoltagePhaseSelector_CH3		: UINT;											//Voltage Phase Selector 1/2/3 for Channel 3
	uiVoltagePhaseSelector_CH4		: UINT;											//Voltage Phase Selector 1/2/3 for Channel 4
	uiVoltagePhaseSelector_CH5		: UINT;											//Voltage Phase Selector 1/2/3 for Channel 5
	uiVoltagePhaseSelector_CH6		: UINT;											//Voltage Phase Selector 1/2/3 for Channel 6 
END_VAR
VAR_OUTPUT
	m_Busy: BOOL;
	m_CoE_Write_done: BOOL;
	m_Error: bool;
	udint_GetAMSNetID_Error: UDINT;
	udint_WriteCoE_Error: UDINT;
END_VAR
VAR
	i_State	:UINT:=1;
	fb_GetAMSNetID	:FB_GetLocalAmsNetId;
  	fb_coe_write          : FB_EcCoESdoWrite; // Function Block for writing in CoE


	r_trig_Start: R_trig;
	i_errorCount: INT;
	i_AMSNetID_ReadOut_Succesfull: INT;
	str_AMSNetID: STRING(30);
 	nValue     : UdINT ; (* variable to be written to the CoE Object *)
 	
	i_CoE_Write_Succesfull: INT;
	udint_Value: UDINT;
	real_Value: REAL;

END_VAR


r_trig_Start(Clk := m_start);

CASE i_State OF
	1: 		// wait for start
	IF r_trig_Start.Q THEN
		i_State := i_State+1;
		m_CoE_Write_done := FALSE;
		m_Busy := TRUE;
		m_Error := FALSE;
	END_IF

	2:		// read out ams net ID	
	fb_GetAMSNetID.bExecute := TRUE;
	i_State := i_State+1;
	
	3: 		// wait for read ot
	IF fb_GetAMSNetID.bBusy = FALSE AND NOT fb_GetAMSNetID.bError = TRUE THEN
		fb_GetAMSNetID.bExecute := FALSE;
		i_AMSNetID_ReadOut_Succesfull := i_AMSNetID_ReadOut_Succesfull+1;
		i_State := i_State+1;
	ELSIF fb_GetAMSNetID.bError = TRUE THEN
		fb_GetAMSNetID.bExecute := FALSE;
		i_State := 100;
	END_IF
	
	4: 		// read out AMS Net ID done, convert received data
	str_AMSNetID := concat(BYTE_TO_STRING(fb_GetAMSNetID.AddrBytes[0]),'.');
	str_AMSNetID := concat(str_AMSNetID,BYTE_TO_STRING(fb_GetAMSNetID.AddrBytes[1]));
	str_AMSNetID := concat(str_AMSNetID,'.');	
	str_AMSNetID := concat(str_AMSNetID,BYTE_TO_STRING(fb_GetAMSNetID.AddrBytes[2]));
	str_AMSNetID := concat(str_AMSNetID,'.');
	str_AMSNetID := concat(str_AMSNetID,BYTE_TO_STRING(fb_GetAMSNetID.AddrBytes[3]));
	str_AMSNetID := concat(str_AMSNetID,'.3.1');
	
	i_State := 10;

	10: 	// write channel 1 phase Selector
	fb_coe_write.bExecute 	:= TRUE;
	fb_coe_write.nIndex		:= 16#8000;
	fb_coe_write.nSubIndex	:= 16#11; 
	udint_Value 			:= UINT_TO_UDINT(uiVoltagePhaseSelector_CH1);
	fb_coe_write.pSrcBuf	:= ADR(udint_Value);
	fb_coe_write.cbBufLen	:= SIZEOF(udint_Value);
	i_State := i_State+1;
	
	11: 	// wait for done or error
	IF NOT fb_coe_write.bBusy AND NOT fb_coe_write.bError THEN
		fb_coe_write.bExecute 	:= FALSE;
		i_CoE_Write_Succesfull := i_CoE_Write_Succesfull+1;
		i_State := i_State+1;
	ELSIF fb_coe_write.bError THEN
		fb_coe_write.bExecute 	:= FALSE;
		i_State := 100;
	END_IF

	12:		// wait 
	i_State := 20;
	
	20: 	// write channel 2 phase Selector
	fb_coe_write.bExecute 	:= TRUE;
	fb_coe_write.nIndex		:= 16#8010;
	fb_coe_write.nSubIndex	:= 16#11; 
	udint_Value 			:= UINT_TO_UDINT(uiVoltagePhaseSelector_CH2);
	fb_coe_write.pSrcBuf	:= ADR(udint_Value);
	fb_coe_write.cbBufLen	:= SIZEOF(udint_Value);
	i_State := i_State+1;
	
	21: 	// wait for done or error
	IF NOT fb_coe_write.bBusy AND NOT fb_coe_write.bError THEN
		fb_coe_write.bExecute 	:= FALSE;
		i_CoE_Write_Succesfull := i_CoE_Write_Succesfull+1;
		i_State := i_State+1;
	ELSIF fb_coe_write.bError THEN
		fb_coe_write.bExecute 	:= FALSE;
		i_State := 100;
	END_IF

	22:		// wait 
	i_State := 30;

	30: 	// write channel 3 phase Selector
	fb_coe_write.bExecute 	:= TRUE;
	fb_coe_write.nIndex		:= 16#8020;
	fb_coe_write.nSubIndex	:= 16#11; 
	udint_Value 			:= UINT_TO_UDINT(uiVoltagePhaseSelector_CH3);
	fb_coe_write.pSrcBuf	:= ADR(udint_Value);
	fb_coe_write.cbBufLen	:= SIZEOF(udint_Value);
	i_State := i_State+1;
	
	31: 	// wait for done or error
	IF NOT fb_coe_write.bBusy AND NOT fb_coe_write.bError THEN
		fb_coe_write.bExecute 	:= FALSE;
		i_CoE_Write_Succesfull := i_CoE_Write_Succesfull+1;
		i_State := i_State+1;
	ELSIF fb_coe_write.bError THEN
		fb_coe_write.bExecute 	:= FALSE;
		i_State := 100;
	END_IF

	32:		// wait 
	i_State := 40;
	
	40: 	// write channel 4 phase Selector
	fb_coe_write.bExecute 	:= TRUE;
	fb_coe_write.nIndex		:= 16#8030;
	fb_coe_write.nSubIndex	:= 16#11; 
	udint_Value 			:= UINT_TO_UDINT(uiVoltagePhaseSelector_CH4);
	fb_coe_write.pSrcBuf	:= ADR(udint_Value);
	fb_coe_write.cbBufLen	:= SIZEOF(udint_Value);
	i_State := i_State+1;
	
	41: 	// wait for done or error
	IF NOT fb_coe_write.bBusy AND NOT fb_coe_write.bError THEN
		fb_coe_write.bExecute 	:= FALSE;
		i_CoE_Write_Succesfull := i_CoE_Write_Succesfull+1;
		i_State := i_State+1;
	ELSIF fb_coe_write.bError THEN
		fb_coe_write.bExecute 	:= FALSE;
		i_State := 100;
	END_IF

	42:		// wait 
	i_State := 50;		

	50: 	// write channel 5 phase Selector
	fb_coe_write.bExecute 	:= TRUE;
	fb_coe_write.nIndex		:= 16#8040;
	fb_coe_write.nSubIndex	:= 16#11; 
	udint_Value 			:= UINT_TO_UDINT(uiVoltagePhaseSelector_CH5);
	fb_coe_write.pSrcBuf	:= ADR(udint_Value);
	fb_coe_write.cbBufLen	:= SIZEOF(udint_Value);
	i_State := i_State+1;
	
	51: 	// wait for done or error
	IF NOT fb_coe_write.bBusy AND NOT fb_coe_write.bError THEN
		fb_coe_write.bExecute 	:= FALSE;
		i_CoE_Write_Succesfull := i_CoE_Write_Succesfull+1;
		i_State := i_State+1;
	ELSIF fb_coe_write.bError THEN
		fb_coe_write.bExecute 	:= FALSE;
		i_State := 100;
	END_IF

	52:		// wait 
	i_State := 60;		

	60: 	// write channel 6 phase Selector
	fb_coe_write.bExecute 	:= TRUE;
	fb_coe_write.nIndex		:= 16#8050;
	fb_coe_write.nSubIndex	:= 16#11; 
	udint_Value 			:= UINT_TO_UDINT(uiVoltagePhaseSelector_CH6);
	fb_coe_write.pSrcBuf	:= ADR(udint_Value);
	fb_coe_write.cbBufLen	:= SIZEOF(udint_Value);
	i_State := i_State+1;
	
	61: 	// wait for done or error
	IF NOT fb_coe_write.bBusy AND NOT fb_coe_write.bError THEN
		fb_coe_write.bExecute 	:= FALSE;
		i_CoE_Write_Succesfull := i_CoE_Write_Succesfull+1;
		i_State := i_State+1;
	ELSIF fb_coe_write.bError THEN
		fb_coe_write.bExecute 	:= FALSE;
		i_State := 100;
	END_IF

	62:		// wait 
	m_CoE_Write_done := TRUE;
	m_Busy := FALSE;
	i_State := 1;		
	
	100: 	//error state
	i_errorCount := i_errorCount +1;
	udint_GetAMSNetID_Error := fb_GetAMSNetID.nErrId;
	udint_WriteCoE_Error := fb_coe_write.nErrId;
	m_Busy := FALSE;
	m_Error := true;
	i_State := 1;

END_CASE


fb_GetAMSNetID(
	bExecute:= , 
	tTimeOut:= T#2S, 
	bBusy=> , 
	bError=> , 
	nErrId=> , 
	AddrString=> , 
	AddrBytes=> );
	
fb_coe_write(
	sNetId:= str_AMSNetID, 
	nSlaveAddr:= nSlaveAddr, 
	nSubIndex:= , 
	nIndex:= , 
    pSrcBuf    := ,
    cbBufLen   := ,
	bExecute:= , 
	tTimeout:= T#2S , 
	bBusy=> , 
	bError=> , 
	nErrId=> );

END_FUNCTION_BLOCK

// ---- FBs/FB_CoE_EL3443.TcPOU
FUNCTION_BLOCK FB_CoE_EL3443
VAR_INPUT
	m_start: BOOL;
	nSlaveAddr	:UINT;
	uiCurrentTransformerRatio		: UINT;											//CT Ratio
END_VAR
VAR_OUTPUT
	m_Busy: BOOL;
	m_CoE_Write_done: BOOL;
	m_Error: bool;
	udint_GetAMSNetID_Error: UDINT;
	udint_WriteCoE_Error: UDINT;
END_VAR
VAR
	i_State	:UINT:=1;
	fb_GetAMSNetID	:FB_GetLocalAmsNetId;
  	fb_coe_write          : FB_EcCoESdoWrite; // Function Block for writing in CoE


	r_trig_Start: R_trig;
	i_errorCount: INT;
	i_AMSNetID_ReadOut_Succesfull: INT;
	str_AMSNetID: STRING(30);
 	real_Value     : REAL ; (* variable to be written to the CoE Object *)
 	
	i_CoE_Write_Succesfull: INT;

	real_Current_Min_Warning 	: REAL	:=-100;
	real_Current_Min_Error 		: REAL	:=-120;
	real_Current_Max_Warning 	: REAL	:= 100;
	real_Current_Max_Error 		: REAL	:= 120;
	


END_VAR


r_trig_Start(Clk := m_start);

CASE i_State OF
	1: 		// wait for start
	IF r_trig_Start.Q THEN
		i_State := i_State+1;
		m_CoE_Write_done := FALSE;
		m_Busy := TRUE;
		m_Error := FALSE;
	END_IF

	2:		// read out ams net ID	
	fb_GetAMSNetID.bExecute := TRUE;
	i_State := i_State+1;
	
	3: 		// wait for read out
	IF fb_GetAMSNetID.bBusy = FALSE AND NOT fb_GetAMSNetID.bError = TRUE THEN
		fb_GetAMSNetID.bExecute := FALSE;
		i_AMSNetID_ReadOut_Succesfull := i_AMSNetID_ReadOut_Succesfull+1;
		i_State := i_State+1;
	ELSIF fb_GetAMSNetID.bError = TRUE THEN
		fb_GetAMSNetID.bExecute := FALSE;
		i_State := 100;
	END_IF
	
	4: 		// read out AMS Net ID done, convert received data
	str_AMSNetID := concat(BYTE_TO_STRING(fb_GetAMSNetID.AddrBytes[0]),'.');
	str_AMSNetID := concat(str_AMSNetID,BYTE_TO_STRING(fb_GetAMSNetID.AddrBytes[1]));
	str_AMSNetID := concat(str_AMSNetID,'.');	
	str_AMSNetID := concat(str_AMSNetID,BYTE_TO_STRING(fb_GetAMSNetID.AddrBytes[2]));
	str_AMSNetID := concat(str_AMSNetID,'.');
	str_AMSNetID := concat(str_AMSNetID,BYTE_TO_STRING(fb_GetAMSNetID.AddrBytes[3]));
	str_AMSNetID := concat(str_AMSNetID,'.3.1');
	
	i_State := 10;

	10: 	// write channel 1 
	fb_coe_write.bExecute 	:= TRUE;
	fb_coe_write.nIndex		:= 16#8000;
	fb_coe_write.nSubIndex	:= 16#12; 
	real_Value 			:= UINT_TO_REAL(uiCurrentTransformerRatio);
	fb_coe_write.pSrcBuf	:= ADR(real_Value);
	fb_coe_write.cbBufLen	:= SIZEOF(real_Value);
	i_State := i_State+1;
	
	11: 	// wait for done or error
	IF NOT fb_coe_write.bBusy AND NOT fb_coe_write.bError THEN
		fb_coe_write.bExecute 	:= FALSE;
		i_CoE_Write_Succesfull := i_CoE_Write_Succesfull+1;
		i_State := i_State+1;
	ELSIF fb_coe_write.bError THEN
		fb_coe_write.bExecute 	:= FALSE;
		i_State := 100;
	END_IF

	12:		// wait 
	i_State := 20;
	
	20: 	// write channel 2 
	fb_coe_write.bExecute 	:= TRUE;
	fb_coe_write.nIndex		:= 16#8010;
	fb_coe_write.nSubIndex	:= 16#12; 
	real_Value 			:= UINT_TO_REAL(uiCurrentTransformerRatio);
	fb_coe_write.pSrcBuf	:= ADR(real_Value);
	fb_coe_write.cbBufLen	:= SIZEOF(real_Value);
	i_State := i_State+1;
	
	21: 	// wait for done or error
	IF NOT fb_coe_write.bBusy AND NOT fb_coe_write.bError THEN
		fb_coe_write.bExecute 	:= FALSE;
		i_CoE_Write_Succesfull := i_CoE_Write_Succesfull+1;
		i_State := i_State+1;
	ELSIF fb_coe_write.bError THEN
		fb_coe_write.bExecute 	:= FALSE;
		i_State := 100;
	END_IF

	22:		// wait 
	i_State := 30;

	30: 	// write channel 3 
	fb_coe_write.bExecute 	:= TRUE;
	fb_coe_write.nIndex		:= 16#8020;
	fb_coe_write.nSubIndex	:= 16#12; 
	real_Value 			:= UINT_TO_REAL(uiCurrentTransformerRatio);
	fb_coe_write.pSrcBuf	:= ADR(real_Value);
	fb_coe_write.cbBufLen	:= SIZEOF(real_Value);
	i_State := i_State+1;
	
	31: 	// wait for done or error
	IF NOT fb_coe_write.bBusy AND NOT fb_coe_write.bError THEN
		fb_coe_write.bExecute 	:= FALSE;
		i_CoE_Write_Succesfull := i_CoE_Write_Succesfull+1;
		i_State := i_State+1;
	ELSIF fb_coe_write.bError THEN
		fb_coe_write.bExecute 	:= FALSE;
		i_State := 100;
	END_IF

	32:		// wait 
	i_State := 40;		

	40: 	// write Channel 1 current guard min error 
	fb_coe_write.bExecute 	:= TRUE;
	fb_coe_write.nIndex		:= 16#8001;
	fb_coe_write.nSubIndex	:= 16#15; 
	real_Value 			:= (real_Current_Min_Error);
	fb_coe_write.pSrcBuf	:= ADR(real_Value);
	fb_coe_write.cbBufLen	:= SIZEOF(real_Value);
	i_State := i_State+1;
	
	41: 	// wait for done or error
	IF NOT fb_coe_write.bBusy AND NOT fb_coe_write.bError THEN
		fb_coe_write.bExecute 	:= FALSE;
		i_CoE_Write_Succesfull := i_CoE_Write_Succesfull+1;
		i_State := i_State+1;
	ELSIF fb_coe_write.bError THEN
		fb_coe_write.bExecute 	:= FALSE;
		i_State := 100;
	END_IF
	
	42:		// wait 
	i_State := i_State+1;		

	43: 	// write Channel 1 current guard min warning 
	fb_coe_write.bExecute 	:= TRUE;
	fb_coe_write.nIndex		:= 16#8001;
	fb_coe_write.nSubIndex	:= 16#16; 
	real_Value 			:= (real_Current_Min_Warning);
	fb_coe_write.pSrcBuf	:= ADR(real_Value);
	fb_coe_write.cbBufLen	:= SIZEOF(real_Value);
	i_State := i_State+1;
	
	44: 	// wait for done or error
	IF NOT fb_coe_write.bBusy AND NOT fb_coe_write.bError THEN
		fb_coe_write.bExecute 	:= FALSE;
		i_CoE_Write_Succesfull := i_CoE_Write_Succesfull+1;
		i_State := i_State+1;
	ELSIF fb_coe_write.bError THEN
		fb_coe_write.bExecute 	:= FALSE;
		i_State := 100;
	END_IF

	45:		// wait 
	i_State := i_State+1;		

	46: 	// write Channel 1 current guard max warning 
	fb_coe_write.bExecute 	:= TRUE;
	fb_coe_write.nIndex		:= 16#8001;
	fb_coe_write.nSubIndex	:= 16#17; 
	real_Value 			:= (real_Current_Max_Warning);
	fb_coe_write.pSrcBuf	:= ADR(real_Value);
	fb_coe_write.cbBufLen	:= SIZEOF(real_Value);
	i_State := i_State+1;
	
	47: 	// wait for done or error
	IF NOT fb_coe_write.bBusy AND NOT fb_coe_write.bError THEN
		fb_coe_write.bExecute 	:= FALSE;
		i_CoE_Write_Succesfull := i_CoE_Write_Succesfull+1;
		i_State := i_State+1;
	ELSIF fb_coe_write.bError THEN
		fb_coe_write.bExecute 	:= FALSE;
		i_State := 100;
	END_IF
	
	48:		// wait 
	i_State := i_State+1;		

	49: 	// write Channel 1 current guard max error 
	fb_coe_write.bExecute 	:= TRUE;
	fb_coe_write.nIndex		:= 16#8001;
	fb_coe_write.nSubIndex	:= 16#18; 
	real_Value 			:= (real_Current_Max_Error);
	fb_coe_write.pSrcBuf	:= ADR(real_Value);
	fb_coe_write.cbBufLen	:= SIZEOF(real_Value);
	i_State := i_State+1;
	
	50: 	// wait for done or error
	IF NOT fb_coe_write.bBusy AND NOT fb_coe_write.bError THEN
		fb_coe_write.bExecute 	:= FALSE;
		i_CoE_Write_Succesfull := i_CoE_Write_Succesfull+1;
		i_State := i_State+1;
	ELSIF fb_coe_write.bError THEN
		fb_coe_write.bExecute 	:= FALSE;
		i_State := 100;
	END_IF

	51:		// wait 
	i_State := i_State+1;	

	52: 	// write Channel 2 current guard min error 
	fb_coe_write.bExecute 	:= TRUE;
	fb_coe_write.nIndex		:= 16#8011;
	fb_coe_write.nSubIndex	:= 16#15; 
	real_Value 			:= (real_Current_Min_Error);
	fb_coe_write.pSrcBuf	:= ADR(real_Value);
	fb_coe_write.cbBufLen	:= SIZEOF(real_Value);
	i_State := i_State+1;
	
	53: 	// wait for done or error
	IF NOT fb_coe_write.bBusy AND NOT fb_coe_write.bError THEN
		fb_coe_write.bExecute 	:= FALSE;
		i_CoE_Write_Succesfull := i_CoE_Write_Succesfull+1;
		i_State := i_State+1;
	ELSIF fb_coe_write.bError THEN
		fb_coe_write.bExecute 	:= FALSE;
		i_State := 100;
	END_IF
	
	54:		// wait 
	i_State := i_State+1;		

	55: 	// write Channel 2 current guard min warning 
	fb_coe_write.bExecute 	:= TRUE;
	fb_coe_write.nIndex		:= 16#8011;
	fb_coe_write.nSubIndex	:= 16#16; 
	real_Value 			:= (real_Current_Min_Warning);
	fb_coe_write.pSrcBuf	:= ADR(real_Value);
	fb_coe_write.cbBufLen	:= SIZEOF(real_Value);
	i_State := i_State+1;
	
	56: 	// wait for done or error
	IF NOT fb_coe_write.bBusy AND NOT fb_coe_write.bError THEN
		fb_coe_write.bExecute 	:= FALSE;
		i_CoE_Write_Succesfull := i_CoE_Write_Succesfull+1;
		i_State := i_State+1;
	ELSIF fb_coe_write.bError THEN
		fb_coe_write.bExecute 	:= FALSE;
		i_State := 100;
	END_IF

	57:		// wait 
	i_State := i_State+1;		

	58: 	// write Channel 2 current guard max warning 
	fb_coe_write.bExecute 	:= TRUE;
	fb_coe_write.nIndex		:= 16#8011;
	fb_coe_write.nSubIndex	:= 16#17; 
	real_Value 			:= (real_Current_Max_Warning);
	fb_coe_write.pSrcBuf	:= ADR(real_Value);
	fb_coe_write.cbBufLen	:= SIZEOF(real_Value);
	i_State := i_State+1;
	
	59: 	// wait for done or error
	IF NOT fb_coe_write.bBusy AND NOT fb_coe_write.bError THEN
		fb_coe_write.bExecute 	:= FALSE;
		i_CoE_Write_Succesfull := i_CoE_Write_Succesfull+1;
		i_State := i_State+1;
	ELSIF fb_coe_write.bError THEN
		fb_coe_write.bExecute 	:= FALSE;
		i_State := 100;
	END_IF
	
	60:		// wait 
	i_State := i_State+1;		

	61: 	// write Channel 2 current guard max error 
	fb_coe_write.bExecute 	:= TRUE;
	fb_coe_write.nIndex		:= 16#8011;
	fb_coe_write.nSubIndex	:= 16#18; 
	real_Value 			:= (real_Current_Max_Error);
	fb_coe_write.pSrcBuf	:= ADR(real_Value);
	fb_coe_write.cbBufLen	:= SIZEOF(real_Value);
	i_State := i_State+1;
	
	62: 	// wait for done or error
	IF NOT fb_coe_write.bBusy AND NOT fb_coe_write.bError THEN
		fb_coe_write.bExecute 	:= FALSE;
		i_CoE_Write_Succesfull := i_CoE_Write_Succesfull+1;
		i_State := i_State+1;
	ELSIF fb_coe_write.bError THEN
		fb_coe_write.bExecute 	:= FALSE;
		i_State := 100;
	END_IF
	
	63:		// wait 
	i_State := i_State+1;	

	64: 	// write Channel 3 current guard min error 
	fb_coe_write.bExecute 	:= TRUE;
	fb_coe_write.nIndex		:= 16#8021;
	fb_coe_write.nSubIndex	:= 16#15; 
	real_Value 			:= (real_Current_Min_Error);
	fb_coe_write.pSrcBuf	:= ADR(real_Value);
	fb_coe_write.cbBufLen	:= SIZEOF(real_Value);
	i_State := i_State+1;
	
	65: 	// wait for done or error
	IF NOT fb_coe_write.bBusy AND NOT fb_coe_write.bError THEN
		fb_coe_write.bExecute 	:= FALSE;
		i_CoE_Write_Succesfull := i_CoE_Write_Succesfull+1;
		i_State := i_State+1;
	ELSIF fb_coe_write.bError THEN
		fb_coe_write.bExecute 	:= FALSE;
		i_State := 100;
	END_IF
	
	66:		// wait 
	i_State := i_State+1;		

	67: 	// write Channel 3 current guard min warning 
	fb_coe_write.bExecute 	:= TRUE;
	fb_coe_write.nIndex		:= 16#8021;
	fb_coe_write.nSubIndex	:= 16#16; 
	real_Value 			:= (real_Current_Min_Warning);
	fb_coe_write.pSrcBuf	:= ADR(real_Value);
	fb_coe_write.cbBufLen	:= SIZEOF(real_Value);
	i_State := i_State+1;
	
	68: 	// wait for done or error
	IF NOT fb_coe_write.bBusy AND NOT fb_coe_write.bError THEN
		fb_coe_write.bExecute 	:= FALSE;
		i_CoE_Write_Succesfull := i_CoE_Write_Succesfull+1;
		i_State := i_State+1;
	ELSIF fb_coe_write.bError THEN
		fb_coe_write.bExecute 	:= FALSE;
		i_State := 100;
	END_IF

	69:		// wait 
	i_State := i_State+1;		

	70: 	// write Channel 3 current guard max warning 
	fb_coe_write.bExecute 	:= TRUE;
	fb_coe_write.nIndex		:= 16#8021;
	fb_coe_write.nSubIndex	:= 16#17; 
	real_Value 			:= (real_Current_Max_Warning);
	fb_coe_write.pSrcBuf	:= ADR(real_Value);
	fb_coe_write.cbBufLen	:= SIZEOF(real_Value);
	i_State := i_State+1;
	
	71: 	// wait for done or error
	IF NOT fb_coe_write.bBusy AND NOT fb_coe_write.bError THEN
		fb_coe_write.bExecute 	:= FALSE;
		i_CoE_Write_Succesfull := i_CoE_Write_Succesfull+1;
		i_State := i_State+1;
	ELSIF fb_coe_write.bError THEN
		fb_coe_write.bExecute 	:= FALSE;
		i_State := 100;
	END_IF
	
	72:		// wait 
	i_State := i_State+1;		

	73: 	// write Channel 3 current guard max warning 
	fb_coe_write.bExecute 	:= TRUE;
	fb_coe_write.nIndex		:= 16#8021;
	fb_coe_write.nSubIndex	:= 16#18; 
	real_Value 			:= (real_Current_Max_Error);
	fb_coe_write.pSrcBuf	:= ADR(real_Value);
	fb_coe_write.cbBufLen	:= SIZEOF(real_Value);
	i_State := i_State+1;
	
	74: 	// wait for done or error
	IF NOT fb_coe_write.bBusy AND NOT fb_coe_write.bError THEN
		fb_coe_write.bExecute 	:= FALSE;
		i_CoE_Write_Succesfull := i_CoE_Write_Succesfull+1;
		i_State := i_State+1;
	ELSIF fb_coe_write.bError THEN
		fb_coe_write.bExecute 	:= FALSE;
		i_State := 100;
	END_IF	
	
	75:		// wait *)
	m_CoE_Write_done := TRUE;
	m_Busy := FALSE;
	i_State := 1;	
	
	100: 	//error state
	i_errorCount := i_errorCount +1;
	udint_GetAMSNetID_Error := fb_GetAMSNetID.nErrId;
	udint_WriteCoE_Error := fb_coe_write.nErrId;
	m_Busy := FALSE;
	m_Error := true;
	i_State := 1;

END_CASE


fb_GetAMSNetID(
	bExecute:= , 
	tTimeOut:= T#2S, 
	bBusy=> , 
	bError=> , 
	nErrId=> , 
	AddrString=> , 
	AddrBytes=> );
	
fb_coe_write(
	sNetId:= str_AMSNetID, 
	nSlaveAddr:= nSlaveAddr, 
	nSubIndex:= , 
	nIndex:= , 
    pSrcBuf    := ,
    cbBufLen   := ,
	bExecute:= , 
	tTimeout:= T#2S , 
	bBusy=> , 
	bError=> , 
	nErrId=> );

END_FUNCTION_BLOCK

// ---- FBs/FB_EM_Beckhoff_EL3443.TcPOU
FUNCTION_BLOCK FB_EM_Beckhoff_EL3443
VAR_INPUT
	bEnable							: BOOL;											//Enable the function
 	bInvers_CH1						: BOOL;											//Invert the Output data from Channel 1 
	bInvers_CH2						: BOOL;											//Invert the Output data from Channel 2 
	bInvers_CH3						: BOOL;											//Invert the Output data from Channel 3
	uiCurrentTransformerRatio		: UINT;											//Current Transformer Ratio  
	nSlaveAddr						: UINT;											//EtherCat Slave ID	
 	stEL3443_IO 						: MDP5001_341_7CD731EE;
END_VAR
VAR_OUTPUT
   	pDpmData 						: POINTER TO ARRAY[1..20] OF UDINT;
	stDataEMPower					: ST_ElectricMeter_Output_Power;				//Output structure with Data from Electric Meter (Power Data) 
	stDataEMCounter					: ST_ElectricMeter_Output_Counter;				//Output structure with Data from Electric Meter (Counter Data) 
	stDataEMPowerRealTime			: ST_ElectricMeter_Output_Power;				//Output structure with Data from Electric Meter (Power Data RealTime)
	stDataEMCounterRealTime			: ST_ElectricMeter_Output_Counter;				//Output structure with Data from Electric Meter (Counter Data RealTime) 
END_VAR
VAR
	fbEM							: FB_ElectricMeter;								//Electric Meter Function
	fbEnergyCounter					: FB_EnergyCounter;								//FB energy Counter, because the KL3403 has no nice logic for the Energy value
	fbEL3443DPM 					: FB_EL3443_DPM;
	
	fb_WriteCOE_EL3443	:FB_Coe_EL3443;	
	m_COE_Done: BOOL;
	uiCurrentTransformerRatio_old		: UINT;											//Current Transformer Ratio  
	f_trig_Busy: f_trig;

	
	timDissableFunctions			: TON;											//Timer to dissable the Function after Lynus_Standards.Constants_General.tTimeDissableLynusFunctions Days without connection to the Lynus Cloud
	timResetConnectionOnGVL			: TON;											//Timer to try reset the connection Flag on the GVL. (When somebody delete the Connection Function and make only a onlinechange)
	timSetCounterValues				: TON;											//Timer to set the counter values from the KL3403 Function to the EM Function
	arrPD							: ARRAY[1..7] OF FB_PersistentData_Number;		//Function to save persistent data
	byWaitInStep					: BYTE;											//Wait in Step before start to clean data on PLC
	iStateGVLData					: INT;											//State machine to handle the data on the GVL
	diCounterForGVL					: DINT;											//Counter to clean old data on GVL
	real_Multiplier_CH1: REAL;
	real_Multiplier_CH2: REAL;
	real_Multiplier_CH3: REAL;
END_VAR

//Creator : Stefan Lackner
//Company : EfficientIO
//Date : xx.09.2023
//Version : 1.0.0.0


//With this function is possible to read out all Information from a EL3446

//NOTE for diNr.....Designation => 
//_IN = Here Data come in from other Functions or go out to other functions about the GVL
//_OUT = Here Data go out to other functions about the GVL



(*-------------------------------------------------------------Service from Backend is ready and check the connection to backen for dissabel/enable Function---------------------------------------------------------------*)

//Try to reset the variable for connection on the GVL. When all is normal then the Lynus Mqtt connection function set this variable to true in the next cycle
//When we have no connection to the backend then after Lynus_Standards.Constants_General.tTimeDissableLynusFunctions days the Function is dissabled with all of his functionalities
timResetConnectionOnGVL(IN:= NOT timResetConnectionOnGVL.Q, PT:= T#1H, Q=> , ET=> );
IF timResetConnectionOnGVL.Q THEN 
	Lynus_Standards.GVL_Communicator.bStateConnectionToEnableFunctions := FALSE; 
END_IF
IF NOT Lynus_Standards.GVL_Communicator.bStateConnectionToEnableFunctions THEN 
	timDissableFunctions.IN := TRUE; 
ELSE 
	timDissableFunctions.IN := FALSE; 
END_IF  
timDissableFunctions(IN:= , PT:= Lynus_Standards.Constants_General.tTimeDissableLynusFunctions, Q=> , ET=> );

// limit inputs
uiCurrentTransformerRatio	 := LIMIT (1,uiCurrentTransformerRatio,10000);


(*----------------------------------------------------------------------------------------EL3446 Communication----------------------------------------------------------------------------------------------*)
// write CoE values for phase selector

IF 	NOT m_COE_Done OR 	uiCurrentTransformerRatio <> uiCurrentTransformerRatio_old THEN
	fb_WriteCOE_EL3443.m_start := TRUE;
	m_COE_Done := TRUE;
	 uiCurrentTransformerRatio_old := uiCurrentTransformerRatio;
END_IF
f_trig_Busy(CLK := fb_WriteCOE_EL3443.m_Busy );
IF f_trig_Busy.Q AND (fb_WriteCOE_EL3443.m_CoE_Write_done OR fb_WriteCOE_EL3443.m_Error) THEN 
	fb_WriteCOE_EL3443.m_start := FALSE;
END_IF

fb_WriteCOE_EL3443(
	m_start:= , 
	nSlaveAddr:= nSlaveAddr, 
	uiCurrentTransformerRatio:= uiCurrentTransformerRatio, 
	m_Busy=> , 
	m_CoE_Write_done=> , 
	m_Error=> , 
	udint_GetAMSNetID_Error=> , 
	udint_WriteCoE_Error=> );



fbEL3443DPM(
	bEnable:= TRUE, 
	stEL3443_IO:= stEL3443_IO , 
	stStatusTotal=> , 
	stStatusPhase_L1=> , 
	stStatusPhase_L2=> , 
	stStatusPhase_L3=> , 
	stVariantValues=> , 
	pDpmData=> pDpmData, 
	bError=> );






//Invert the Output data, because it is possible that the current transformers have been mounted in different mounting positions.
IF NOT bInvers_CH1 THEN
	real_Multiplier_CH1 := 1;
ELSE
	real_Multiplier_CH1 := -1;
END_IF
IF NOT bInvers_CH2 THEN
	real_Multiplier_CH2 := 1;
ELSE
	real_Multiplier_CH2 := -1;
END_IF
IF NOT bInvers_CH3 THEN
	real_Multiplier_CH3 := 1;
ELSE
	real_Multiplier_CH3 := -1;
END_IF


//Function
fbEM(
	bEnable:= bEnable AND NOT timDissableFunctions.Q, 
	bError:= , 
	bEnableReadOutFunction:= FALSE, 
	bWriteWithDelay:= TRUE, 
	bPowerDataInvers:= FALSE,
	bReadOutDataDone:= timSetCounterValues.Q,
	iTimeReadOutInterval:= 0, 
	iErrorCode:= , 
	iWarningCode:= , 
	lrTotalCounterEnergy_Consumption:= fbEnergyCounter.lrTotalCounterEnergy_Consumption,
	lrTotalCounterEnergy_Production:= fbEnergyCounter.lrTotalCounterEnergy_Production, 
	lrCounterEnergyT1_Consumption:= fbEnergyCounter.lrCounterEnergyT1_Consumption,
	lrCounterEnergyT2_Consumption:= fbEnergyCounter.lrCounterEnergyT2_Consumption,
	lrCounterEnergyT1_Production:= fbEnergyCounter.lrCounterEnergyT1_Production, 
	lrCounterEnergyT2_Production:= fbEnergyCounter.lrCounterEnergyT2_Production, 
	lrCurrentL1:=  REAL_TO_LREAL(fbEL3443DPM.stEL3443_IO.MDP5001_341_Input.MDP5001_341_L1_Basic_Current ),
	lrVoltageL1N:= REAL_TO_LREAL(fbEL3443DPM.stEL3443_IO.MDP5001_341_Input.MDP5001_341_L1_Basic_Voltage), 
	lrVoltageL1L2:= REAL_TO_LREAL(fbEL3443DPM.stEL3443_IO.MDP5001_341_Input.MDP5001_341_L1_Basic_Voltage * 1.73), 
	lrPowerL1:= REAL_TO_LREAL(fbEL3443DPM.stEL3443_IO.MDP5001_341_Input.MDP5001_341_L1_Power_Active_Power * real_Multiplier_CH1), 
	lrCurrentL2:=  REAL_TO_LREAL(fbEL3443DPM.stEL3443_IO.MDP5001_341_Input.MDP5001_341_L2_Basic_Current),
	lrVoltageL2N:= REAL_TO_LREAL(fbEL3443DPM.stEL3443_IO.MDP5001_341_Input.MDP5001_341_L2_Basic_Voltage), 
	lrVoltageL2L3:= REAL_TO_LREAL(fbEL3443DPM.stEL3443_IO.MDP5001_341_Input.MDP5001_341_L2_Basic_Voltage * 1.73), 
	lrPowerL2:= REAL_TO_LREAL(fbEL3443DPM.stEL3443_IO.MDP5001_341_Input.MDP5001_341_L2_Power_Active_Power  * real_Multiplier_CH2),	
	lrCurrentL3:=  REAL_TO_LREAL(fbEL3443DPM.stEL3443_IO.MDP5001_341_Input.MDP5001_341_L3_Basic_Current),
	lrVoltageL3N:= REAL_TO_LREAL(fbEL3443DPM.stEL3443_IO.MDP5001_341_Input.MDP5001_341_L3_Basic_Voltage), 
	lrVoltageL3L1:= REAL_TO_LREAL(fbEL3443DPM.stEL3443_IO.MDP5001_341_Input.MDP5001_341_L3_Basic_Voltage * 1.73), 
	lrPowerL3:= REAL_TO_LREAL(fbEL3443DPM.stEL3443_IO.MDP5001_341_Input.MDP5001_341_L3_Power_Active_Power * real_Multiplier_CH3),	

